(* CODESYS project kp38822.project

Project tree, tasks and I/O mapping:
  A1_01A : PR-R01, Vira Realtime Ltd, version 5.11.2.0
      settings: NodeName = 'PR-10R'; FtpUser = 'q'; FtpPass = 'q'
      unmapped channels: Service, Clock, Battery, SD, fsTotal, fsFree, Boot, Hardware errors, Kernel errors, Software errors, Source, Time new, Time old, tx, rx, rx_timeout, rx_error, trans_error
    application Application
      libraries: SysMem, * (System); StringUtils, * (System); PR-R01 library, 2.0.0.0 (Vira Realtime Ltd); Standard, * (System); RLT Network utils, * (VIRA Realtime Ltd); RLT Devices Catalogue, * (VIRA Realtime Ltd); RLT Algo blocks implementation, * (VIRA Realtime Ltd); RLT Base IO implementation, * (VIRA Realtime Ltd); SysTimeRtc, * (System); RLT Master Modbus, 1.0.15 (VIRA Realtime Ltd); RLT Slave Modbus, 1.1.0.0 (Vira Realtime Ltd); RLT Slave Modbus TCP, 1.3.0.0 (VIRA Realtime Ltd)
      task TaskMain (cyclic, interval t#100ms, priority 1) calls Main, App104, IP2RS_PRG
      task Daemons (cyclic, interval t#10ms, priority 1) calls DaemonIP, DaemonSerial
      task TaskFlow (cyclic, interval t#50ms, priority 1) calls Devices
      program Main [ST]: Init_Main, Init_Gen, Init_User, Cyclic_In, Cyclic_Main, Cyclic_Out, Cyclic_User, Cyclic_DB, Cyclic_Station
      global variables GVL
      global variables CFG
      global variables CFGCONST
      global variables DBADR
      program App104 [ST]: InRange
      Structs/
        data type station_typ
        data type options_typ
        data type stt_cmd_typ
        data type alarm_typ
        data type sys_mod_typ
        data type server_typ
        data type diag_typ
        pid/
          data type ctrl_cmd_typ
          data type ctrl_flags_typ
          data type ctrl_param_typ
          data type ctrl_input_typ
          data type ctrl_output_typ
          data type line_cmd_typ
          data type line_flags_r_typ
          data type line_act_out
          data type line_act_in
          data type line_cmd_grp_typ
          data type line_flags_f_typ
          data type line_param_f_typ
      Types/
        data type stop_actions
      program Devices [ST]: Init_Gen, Cyclic_Gen, Cyclic_DB
      Enums/
        data type en_stt_mode
        data type en_stt_cfg
        data type en_ctrl_cfg
        data type en_line_action
      Oscat/
        function T_PLC_US [ST]
        function block CTRL_OUT [ST]
        function block FT_PIDWL [ST]
        function CTRL_IN [ST]
        function block FT_PIWL [ST]
        function block FT_DERIV [ST]
        function DEAD_ZONE [ST]
        function block CTRL_PID [ST]
      program DaemonIP [ST]
      program DaemonSerial [ST]
      FUBs/
        function block Controller [ST]
        function block LineMeteringRLT [ST]: Init, _set_mr
        function block LineReducingRLT [ST]: Init, _set_mr
        function block LineGroupRLT [ST]: Init, _next
      global variables DEV
      Devices/
        function block AKP [ST]: Init, FB_init, SetCount
        function block Mercury [ST]: Init, FB_init, SetCount
        function block EK [ST]: Init, FB_init, SetCount
        function block SKP [ST]: Init, FB_init, SetCount
        function block NGK_IPKZ [ST]: Init, FB_init, SetCount
        function block TestGRS [ST]: Init, FB_init, SetCount
        function block VOPETM [ST]: Init, FB_init, SetCount
        function block ERIS [ST]: Init, FB_init, SetCount
      program IP2RS_PRG [ST]
      program PLC_PRG_Slave [ST]
      program POU [ST]
    Time synchronization
        unmapped channels: Source, Time new, Time old
    Ethernet 1
        settings: address = '172.16.26.26'; mask = '255.255.255.240'; gateway = '172.16.26.25'
      Virtual_COM_0 : Virtual COM, Vira Realtime Ltd, version 5.11.2.0
          settings: address = '172.16.26.22'; port = 4000
          unmapped channels: state
      Virtual_COM_1 : Virtual COM, Vira Realtime Ltd, version 5.11.2.0
          settings: address = '172.16.26.22'; port = 4001
          unmapped channels: state
      Virtual_COM_2 : Virtual COM, Vira Realtime Ltd, version 5.11.2.0
          settings: address = '172.16.26.22'; port = 4002
          unmapped channels: state
      Virtual_COM_3 : Virtual COM, Vira Realtime Ltd, version 5.11.2.0
          settings: address = '172.16.26.22'; port = 4003
          unmapped channels: state
      Virtual_COM_4 : Virtual COM, Vira Realtime Ltd, version 5.11.2.0
          settings: address = '172.16.26.22'; port = 4006
          unmapped channels: state
      Virtual_COM_5 : Virtual COM, Vira Realtime Ltd, version 5.11.2.0
          settings: address = '172.16.26.22'; port = 4005
          unmapped channels: state
    Ethernet 2
        settings: address = '172.16.26.100'; mask = '255.255.255.240'; gateway = '0.0.0.0'
    IO Modules
        unmapped channels: tx, rx, rx_timeout, rx_error, trans_error
      A11 : DI32, Vira Realtime Ltd, version 2.22.0.0
          settings: counterState.Group2.Bit7 = TRUE; counterState.Group4.Bit7 = TRUE; fltDI = 0
          input  Application.sys_di[0].di : BOOL  // DI.Group1.DI1
          input  Application.sys_di[1].di : BOOL  // DI.Group1.DI2
          input  Application.sys_di[2].di : BOOL  // DI.Group1.DI3
          input  Application.sys_di[3].di : BOOL  // DI.Group1.DI4
          input  Application.sys_di[4].di : BOOL  // DI.Group1.DI5
          input  Application.sys_di[5].di : BOOL  // DI.Group1.DI6
          input  Application.sys_di[6].di : BOOL  // DI.Group1.DI7
          input  Application.sys_di[7].di : BOOL  // DI.Group1.DI8
          input  Application.sys_di[8].di : BOOL  // DI.Group2.DI9
          input  Application.sys_di[9].di : BOOL  // DI.Group2.DI10
          input  Application.sys_di[10].di : BOOL  // DI.Group2.DI11
          input  Application.sys_di[11].di : BOOL  // DI.Group2.DI12
          input  Application.sys_di[12].di : BOOL  // DI.Group2.DI13
          input  Application.sys_di[13].di : BOOL  // DI.Group2.DI14
          input  Application.sys_di[14].di : BOOL  // DI.Group2.DI15
          input  Application.sys_di[15].di : BOOL  // DI.Group2.DI16
          input  Application.sys_di[16].di : BOOL  // DI.Group3.DI17
          input  Application.sys_di[17].di : BOOL  // DI.Group3.DI18
          input  Application.sys_di[18].di : BOOL  // DI.Group3.DI19
          input  Application.sys_di[19].di : BOOL  // DI.Group3.DI20
          input  Application.sys_di[20].di : BOOL  // DI.Group3.DI21
          input  Application.sys_di[21].di : BOOL  // DI.Group3.DI22
          input  Application.sys_di[22].di : BOOL  // DI.Group3.DI23
          input  Application.sys_di[23].di : BOOL  // DI.Group3.DI24
          input  Application.sys_di[24].di : BOOL  // DI.Group4.DI25
          input  Application.sys_di[25].di : BOOL  // DI.Group4.DI26
          input  Application.sys_di[26].di : BOOL  // DI.Group4.DI27
          input  Application.sys_di[27].di : BOOL  // DI.Group4.DI28
          input  Application.sys_di[28].di : BOOL  // DI.Group4.DI29
          input  Application.sys_di[29].di : BOOL  // DI.Group4.DI30
          input  Application.sys_di[30].di : BOOL  // DI.Group4.DI31
          input  Application.sys_di[31].di : BOOL  // DI.Group4.DI32
          input  Application.impulse_counter : DWORD  // counters.counters
          input  Application.sys_mod[1].ok : BIT  // online
          unmapped channels: DI, counters, tx, rx, rx_timeout, rx_error, trans_error, type, Service, Backline line1, Backline line2
      A12 : DI16/DO16, Vira Realtime Ltd, version 2.22.0.0
          settings: counterState.Group1.Bit0 = FALSE; counterState.Group1.Bit1 = FALSE; counterState.Group1.Bit2 = FALSE; counterState.Group1.Bit3 = FALSE; counterState.Group1.Bit4 = FALSE; counterState.Group1.Bit5 = FALSE; counterState.Group1.Bit6 = FALSE; counterState.Group1.Bit7 = FALSE; counterState.Group2.Bit0 = FALSE; counterState.Group2.Bit1 = FALSE; counterState.Group2.Bit2 = FALSE; counterState.Group2.Bit3 = FALSE; counterState.Group2.Bit4 = FALSE; counterState.Group2.Bit5 = FALSE; counterState.Group2.Bit6 = FALSE; counterState.Group2.Bit7 = TRUE; fltDI = 0
          output Application.sys_do[0].outDO : BOOL  // DO.Group1.DO1
          output Application.sys_do[1].outDO : BOOL  // DO.Group1.DO2
          output Application.sys_do[2].outDO : BOOL  // DO.Group1.DO3
          output Application.sys_do[3].outDO : BOOL  // DO.Group1.DO4
          output Application.sys_do[4].outDO : BOOL  // DO.Group1.DO5
          output Application.sys_do[5].outDO : BOOL  // DO.Group1.DO6
          output Application.sys_do[6].outDO : BOOL  // DO.Group1.DO7
          output Application.sys_do[7].outDO : BOOL  // DO.Group1.DO8
          output Application.sys_do[8].outDO : BOOL  // DO.Group2.DO9
          output Application.sys_do[9].outDO : BOOL  // DO.Group2.DO10
          output Application.sys_do[10].outDO : BOOL  // DO.Group2.DO11
          output Application.sys_do[11].outDO : BOOL  // DO.Group2.DO12
          output Application.sys_do[12].outDO : BOOL  // DO.Group2.DO13
          output Application.sys_do[13].outDO : BOOL  // DO.Group2.DO14
          output Application.sys_do[14].outDO : BOOL  // DO.Group2.DO15
          output Application.sys_do[15].outDO : BOOL  // DO.Group2.DO16
          input  Application.sys_di[32].di : BOOL  // DI.Group1.DI1
          input  Application.sys_di[33].di : BOOL  // DI.Group1.DI2
          input  Application.sys_di[34].di : BOOL  // DI.Group1.DI3
          input  Application.sys_di[35].di : BOOL  // DI.Group1.DI4
          input  Application.sys_di[36].di : BOOL  // DI.Group1.DI5
          input  Application.sys_di[37].di : BOOL  // DI.Group1.DI6
          input  Application.sys_di[38].di : BOOL  // DI.Group1.DI7
          input  Application.sys_di[39].di : BOOL  // DI.Group1.DI8
          input  Application.sys_di[40].di : BOOL  // DI.Group2.DI9
          input  Application.sys_di[41].di : BOOL  // DI.Group2.DI10
          input  Application.sys_di[42].di : BOOL  // DI.Group2.DI11
          input  Application.sys_di[43].di : BOOL  // DI.Group2.DI12
          input  Application.sys_di[44].di : BOOL  // DI.Group2.DI13
          input  Application.sys_di[45].di : BOOL  // DI.Group2.DI14
          input  Application.sys_di[46].di : BOOL  // DI.Group2.DI15
          input  Application.sys_di[47].di : BOOL  // DI.Group2.DI16
          input  Application.sys_do[0].fb_err : BOOL  // DO_bi_err.Group1.Bit0
          input  Application.sys_do[1].fb_err : BOOL  // DO_bi_err.Group1.Bit1
          input  Application.sys_do[2].fb_err : BOOL  // DO_bi_err.Group1.Bit2
          input  Application.sys_do[3].fb_err : BOOL  // DO_bi_err.Group1.Bit3
          input  Application.sys_do[4].fb_err : BOOL  // DO_bi_err.Group1.Bit4
          input  Application.sys_do[5].fb_err : BOOL  // DO_bi_err.Group1.Bit5
          input  Application.sys_do[6].fb_err : BOOL  // DO_bi_err.Group1.Bit6
          input  Application.sys_do[7].fb_err : BOOL  // DO_bi_err.Group1.Bit7
          input  Application.sys_do[8].fb_err : BOOL  // DO_bi_err.Group2.Bit0
          input  Application.sys_do[9].fb_err : BOOL  // DO_bi_err.Group2.Bit1
          input  Application.sys_do[10].fb_err : BOOL  // DO_bi_err.Group2.Bit2
          input  Application.sys_do[11].fb_err : BOOL  // DO_bi_err.Group2.Bit3
          input  Application.sys_do[12].fb_err : BOOL  // DO_bi_err.Group2.Bit4
          input  Application.sys_do[13].fb_err : BOOL  // DO_bi_err.Group2.Bit5
          input  Application.sys_do[14].fb_err : BOOL  // DO_bi_err.Group2.Bit6
          input  Application.sys_do[15].fb_err : BOOL  // DO_bi_err.Group2.Bit7
          input  Application.sys_mod[2].ok : BIT  // online
          unmapped channels: DO, DI, BI, counters, DO_bi_err, tx, rx, rx_timeout, rx_error, trans_error, type, Service, Backline line1, Backline line2
      A13 : AI16, Vira Realtime Ltd, version 2.22.0.0
          input  Application.sys_ai[0].ai : INT  // AI.AI
          input  Application.sys_ai[1].ai : INT  // AI.AI
          input  Application.sys_ai[2].ai : INT  // AI.AI
          input  Application.sys_ai[3].ai : INT  // AI.AI
          input  Application.sys_ai[4].ai : INT  // AI.AI
          input  Application.sys_ai[5].ai : INT  // AI.AI
          input  Application.sys_ai[6].ai : INT  // AI.AI
          input  Application.sys_ai[7].ai : INT  // AI.AI
          input  Application.sys_ai[8].ai : INT  // AI.AI
          input  Application.sys_ai[9].ai : INT  // AI.AI
          input  Application.sys_ai[10].ai : INT  // AI.AI
          input  Application.sys_ai[11].ai : INT  // AI.AI
          input  Application.sys_ai[12].ai : INT  // AI.AI
          input  Application.sys_ai[13].ai : INT  // AI.AI
          input  Application.sys_ai[14].ai : INT  // AI.AI
          input  Application.sys_ai[15].ai : INT  // AI.AI
          input  Application.sys_mod[3].ok : BIT  // online
          unmapped channels: AI, AI_temp, AI_calib, tx, rx, rx_timeout, rx_error, trans_error, type, Service, Backline line1, Backline line2
  libraries: SysTypes Interfaces, 3.5.2.0 (System); SysSocket, 3.5.6.0 (System); SysMem, 3.5.5.0 (System); SysCom, 3.5.5.0 (System); CmpErrors Interfaces, * (System); SysTime, 3.5.5.0 (System); CAA Memory, 3.5.5.0 (CAA Technical Workgroup)
  Client_TCP/
    function block Client_group [ST]: Init, ClientRun, ClientClose, fb_init, fb_exit
    data type Client
    data type ClientState
  Exchange/
    function block Exchange_Buffer [ST]: AddRSMessage, fb_init, GetMessageForRS, ClearByClient, AddIPMessage, CheckIPMessage, Init, GetMessageForIP, DeleteMessage, fb_exit
    data type IP_Buffer
    data type IP_Message
    global variables IP_Message_const
  Serial_port/
    global variables SerialConst
    function block Serial_group [ST]: SlaveRun, fb_exit, fb_init, MasterRun, SlaveProcessRx, Init, MasterProcessRx, FillTxFrame
    data type SerialCfg
    data type Serial
    data type SerialState
    data type SerialHeader
  Server_TCP/
    function block Server_group [ST]: Init, ServerRun, ServerInit, ServerDeinit, fb_exit, fb_init, GetFreeClientIndex, GetClientConfig, ClientClose
    data type SClient
    data type Server
    data type ServerCfg
    data type ClientCfg
  global variables IP_Const
*)

// A1_01A/Application/Types/stop_actions
TYPE stop_actions : ARRAY[0..COUNT_VALVE -1] OF RLTAB.valve_step_actions; END_TYPE

// A1_01A/Application/Structs/station_typ
TYPE station_typ :
STRUCT
//VAR_INPUT
	cfg: UDINT;
	cmd: stt_cmd_typ;
	auto_blocked: BOOL;		// 15	Заблокирован переход в автоматический режим
	
	num_di_valve_dist: UINT;		// привязка напрямую в краны, но нужно указать для точного определения режима
	//num_di_valve_cv: UINT;		// не нужно, привязка напрямую в краны
	num_do_valve_cv: UINT;
	num_di_unit_dist: UINT;
	//num_di_unit_cv: UINT;
	num_do_unit_cv: UINT;
	
	num_di_ack: UINT;		// № ДИ "Квитирование" (если есть)
	num_di_stop_1: UINT;	// № ДИ "Останов 1" (если есть)
	num_di_stop_2: UINT;	// № ДИ "Останов 2" (если есть)
	num_do_sound: UINT;		// № ДО "Звонок" (если есть)
	num_di_sound: UINT;		// № ДИ "Тест звонка" (если есть)
	num_do_alarm: UINT;		// № ДО "Сирена" (если есть)
	num_di_alarm: UINT;		// № ДИ "Тест сирены" (если есть)
	num_do_lamp_fail: UINT;	// № ДО "Лампа авария" (если есть)
	num_do_lamp_alarm: UINT;// № ДО "Лампа предупреждение" (если есть)
	num_do_lamp_fire: UINT;	// № ДО "Лампа пожар" (если есть)
	num_do_lamp_gas: UINT;	// № ДО "Лампа газ" (если есть)
	num_di_lamps: UINT;		// № ДИ "Тест ламп" (если есть)
	num_stop_1: UINT := 0;
	num_stop_2: UINT := 1;
//END_VAR
//VAR_OUTPUT
	time_sys: SysTimeRtc.SysTimeCore.SYSTIME;
	time_plc: SysTimeRtc.RTS_SYSTIMEDATE;
	mode: en_stt_mode;
	mode_auto: BOOL;		// флаг для вычисления режима. не использовать напрямую!
	step_main: UINT;
	user: INT;
	fail_center: ARRAY [0..COUNT_MAX_SERVERS-1] OF BOOL;
	originators: ARRAY [0..COUNT_MAX_SERVERS-1] OF USINT;
	fail_control: BOOL;
	global_imit_di: BOOL;	// 0	Наличие имитации DI
	global_imit_do: BOOL;	// 1	Наличие имитации AI
	global_imit_ai: BOOL;	// 2	Наличие имитации DO
	global_imit_ao: BOOL;	// 3	Наличие имитации AO
	//di_valve_cv: BOOL; \/ // 4	Подготовка ТУ крана
	fail_valve_cv: BOOL;	// 5	Нет подготовки ТУ крана
	//di_unit_cv: BOOL;		// 6	Подготовка ТУ вентилятора
	fail_unit_cv: BOOL;		// 7	Нет подготовки ТУ вентилятора
	sound_blocked: BOOL;	// 8	Блокировка звуковой сигнализации
	global_imit_valve: BOOL;// 9	Обобщенная имитация кранов
	global_imit_unit: BOOL;	// 10	Обобщенная имитация устройств
	global_fail: BOOL;		// 11	Обобщенная авария
	global_warn: BOOL;		// 12	Обобщенное предупреждение
	global_stop: BOOL;		// 13	Идет аварийный останов
	stop_impossible: BOOL;	// 14	Аварийный останов невозможен
	auto_reset: BOOL;		// 16	Автоматический режим остановлен
	err_num: BOOL;
//END_VAR
//VAR
	p_mode: en_stt_mode;
	r_ack: Standard.R_TRIG;
	r_stop_1: Standard.R_TRIG;
	r_stop_2: Standard.R_TRIG;
	//di_valve_dist: BOOL;
	//di_valve_cv: BOOL;
	do_valve_cv: BOOL;
	//di_unit_dist: BOOL;
	//di_unit_cv: BOOL;
	do_unit_cv: BOOL;
	
	di_ack: BOOL;
	di_stop_1: BOOL;
	di_stop_2: BOOL;
	di_sound: BOOL;		// нажатие на кнопку
	do_sound: BOOL;		// логическое
	di_alarm: BOOL;		// нажатие на кнопку
	do_alarm: BOOL;		// логическое
	do_lamp_fail: BOOL;
	do_lamp_alarm: BOOL;
	do_lamp_fire: BOOL;
	do_lamp_gas: BOOL;
	di_lamps: BOOL;		// нажатие на кнопку
	do_lamps: BOOL;		// логическое
//END_VAR
END_STRUCT
END_TYPE

// A1_01A/Application/Structs/options_typ
TYPE options_typ :
STRUCT
	last_group: USINT;
	init: BOOL;
	require_permission: BOOL;
END_STRUCT
END_TYPE

// A1_01A/Application/Enums/en_stt_mode
TYPE en_stt_mode :
(
	MODE_NONE := 0,
	MODE_BUTTON := 1,
	MODE_PART_BUTTON := 2,
	MODE_MANUAL := 3,
	MODE_AUTO := 4
);
END_TYPE

// A1_01A/Application/Enums/en_stt_cfg
TYPE en_stt_cfg :
(
	conf_valve_dist := 0,		// есть общий переключатель "дистанция" для кранов
	conf_valve_cv := 1,			// есть общее ТУ для кранов
	conf_unit_dist := 2,		// есть общий переключатель "дистанция" для устройств
	conf_unit_cv := 3,			// есть общее ТУ для устройств
	conf_sound_block := 4,		// разрешено блокировать звук
	conf_ack := 5,				// есть *физическая* кнопка Квитирование
	conf_stop_1 := 6,			// есть *физическая* кнопка Останов 1
	conf_stop_2 := 7,			// есть *физическая* кнопка Останов 2
	conf_sound := 8,			// есть звонок
	conf_test_sound := 9,		// есть *физическая* кнопка "Тест звонка"
	conf_alarm := 10,			// есть сирена
	conf_test_alarm := 11,		// есть *физическая* кнопка "Тест сирены"
	conf_fail := 12,			// есть лампа "Авария"
	conf_warn := 13,			// есть лампа "Предупреждение"
	conf_fire := 14,			// есть лампа "Пожар"
	conf_gas := 15,				// есть лампа "Газ"
	conf_lamps := 16,			// есть *физическая* кнопка "Тест ламп"
	conf_warn_is_alarm := 17,	// включать аварию по предупреждению
	conf_out_seconds := 18		// выводить секунды в 104
);
END_TYPE

// A1_01A/Application/Structs/stt_cmd_typ
TYPE stt_cmd_typ :
STRUCT
	get_control: BOOL;		// 0	Забрать управление на себя
	mode_auto_off: BOOL;	// 1	Перевести ГРС в автоматизированный режим
	mode_auto_on: BOOL;		// 2	Перевести ГРС в автоматический режим
	mode_auto_reset: BOOL;
	ack_control: BOOL;		// 3	Квитировать ошибку управления
	ack_valves: BOOL;		// 4	Квитирование аварий задвижек
	ack_units: BOOL;		// 5	Квитирование аварий вентиляторов и агрегатов
	ack_alarms: BOOL;		// 6	Квитирование аварий
	reset_imit: BOOL;		// 7	Сброс имитации сигнализации
	imit_valves_on: BOOL;	// 8	Включить имитацию всех задвижек
	imit_valves_off: BOOL;	// 9	Выключить имитацию всех задвижек
	imit_units_on: BOOL;	// 10	Включить имитацию всех вентиляторов
	imit_units_off: BOOL;	// 11	Выключить имитацию всех вентиляторов
	block_sound_on: BOOL;	// 12	Включить блокировку звуковой сигнализации
	block_sound_off: BOOL;	// 13	Выключить блокировку звуковой сигнализации
	sound_on: BOOL;			// 14	Включить звонок
	sound_off: BOOL;		// 15	Выключить звонок
	alarm_on: BOOL;			// 16	Включить сирену
	alarm_off: BOOL;		// 17	Выключить сирену
	lamps_on: BOOL;			// 18	Включить тест ламп
	lamps_off: BOOL;		// 19	Выключить тест ламп
	request_confirm: BOOL;
	request_reject: BOOL;
END_STRUCT
END_TYPE

// A1_01A/Application/Structs/alarm_typ
TYPE alarm_typ :
STRUCT
	active: BOOL;		// сигнал активен
	block: BOOL;		// маска
	imit: BOOL;			// имитация
	type_ack: USINT;	// [0,1] require ack
	cmd_ack: BOOL;
	processed: BOOL;	// обработан
END_STRUCT
END_TYPE

// A1_01A/Application/Structs/sys_mod_typ
TYPE sys_mod_typ :
STRUCT
	name: WSTRING(16);
	id: USINT;
	ok: BOOL;
END_STRUCT
END_TYPE

// Client_TCP/Client
TYPE Client :
STRUCT
	socket			: SysSocket.RTS_IEC_HANDLE;
	to_address		: SOCKADDRESS;
	from_address	: SOCKADDRESS;
	ttl				: UDINT;
	rs_port			: UINT;
	buffer			: POINTER TO Exchange_Buffer;
	rx_data			: ARRAY [0..MSG_SIZE-1] OF BYTE;
	tx_data			: ARRAY [0..MSG_SIZE-1] OF BYTE;
	state			: ClientState;
END_STRUCT
END_TYPE

// Client_TCP/ClientState
TYPE ClientState :
(
	RUN := 0,
	CREATE,
	CONNECT,
	ERROR,
	CLOSE	
) UINT;
END_TYPE

// A1_01A/Application/Structs/server_typ
TYPE server_typ :
STRUCT
    name: WSTRING(16);
    channel: WSTRING(16);
    ip: STRING(16);
    originator: USINT;
    asdu: UINT;
    T1: UINT;
    T2: UINT;
    T3: UINT;
    k: UINT;
    w: UINT;
    port: UINT;
	online: BOOL;
END_STRUCT
END_TYPE

// A1_01A/Application/Structs/pid/ctrl_cmd_typ
TYPE ctrl_cmd_typ :
STRUCT
	manual_on: BOOL;		// ручной режим
	manual_off: BOOL;
	imit_on: BOOL;
	imit_off: BOOL;
	reset: BOOL;			// сброс неисправности
	line_close: BOOL;		// закрыть вместе с линией
END_STRUCT
END_TYPE

// A1_01A/Application/Structs/pid/ctrl_flags_typ
TYPE ctrl_flags_typ :
STRUCT
	mode_dist: BOOL;			// дистанция
	mode_manual: BOOL := 1;		// режим ручного ввода АО
	mode_imit: BOOL;
	mode_discrete: BOOL := 0;	// режим дискретного управления - АО отключается от передачи на модуль
	
	open: BOOL;					// Клапан открыт
	closed: BOOL;				// Клапан закрыт
	ready: BOOL;				// Готов к работе
	block_ao: BOOL;				// Блокировка аналогового управления клапаном
	
	failed: BOOL;				// Неисправность регулирующего клапана
	fail_open: BOOL;			// Регулятор не открылся
	fail_close: BOOL;			// Регулятор не закрылся
END_STRUCT
END_TYPE

// A1_01A/Application/Structs/pid/ctrl_param_typ
TYPE ctrl_param_typ :
STRUCT
	k_p: REAL := 1;
	t_i: REAL := 1;
	t_d: REAL := 0;
	offset: REAL := 0;
	dead_zone: REAL := 0.5;		// зона нечувствительности процесса при регулировании (по значению)
	min_out: REAL := 0;
	max_out: REAL := 100;
	discrepancy: REAL := 0.0;	// значение границы допустимого рассогласования положения крана и регулятора при установлении процесса (в %)
END_STRUCT
END_TYPE

// A1_01A/Application/Enums/en_ctrl_cfg
TYPE en_ctrl_cfg :
(
	discrete_input := 0,
	discrete_output := 1
);
END_TYPE

// A1_01A/Application/Structs/pid/ctrl_input_typ
TYPE ctrl_input_typ :
STRUCT
	act_value: REAL;			// текущее значение параметра, число
	set_value: REAL := 0.0;		// заданное значение параметра, число
	pos_value: REAL;			// текущее положение регулятора, %
	im_pos_value: REAL;			// имитация положение регулятора, %
	hyst_value: REAL := 0.1;	// гистерезис регулятора (дребезг значения положения), %
	man_value: REAL := 0.0;		// ручное управление, %
	
	di_dist: BOOL;				// дистанция
	di_fail: BOOL;				// авария
	
	di_open: BOOL;
	di_closed: BOOL;
END_STRUCT
END_TYPE

// A1_01A/Application/Structs/pid/ctrl_output_typ
TYPE ctrl_output_typ :
STRUCT
	out_value: REAL;			// заданное положение
	err_value: REAL;			// ошибка
	p_part: REAL;
	i_part: REAL;
	d_part: REAL;
	
	do_open: BOOL;
	do_close: BOOL;
	do_stop: BOOL;
END_STRUCT
END_TYPE

// A1_01A/Application/Structs/pid/line_cmd_typ
TYPE line_cmd_typ :
STRUCT
	block_on: BOOL;
	block_off: BOOL;
	manual_on: BOOL;
	manual_off: BOOL;
	//reserve: BOOL;
	reset: BOOL;
	
	open: BOOL;
	close: BOOL;
END_STRUCT
END_TYPE

// A1_01A/Application/Structs/pid/line_flags_r_typ
TYPE line_flags_r_typ :
STRUCT
	open: BOOL;
	closed: BOOL;
	ready: BOOL;				// Готова к работе
	mode_block: BOOL;			// Блокирована
	mode_reserve: BOOL;			// В резерве
	failed: BOOL;				// Неисправность
	fail_block: BOOL;
	err_num: BOOL;
END_STRUCT
END_TYPE

// A1_01A/Application/Enums/en_line_action
TYPE en_line_action :
(
	LA_BUSY := -2,
	LA_ERROR := -1,
	LA_NONE := 0,
	LA_OPEN := 1,
	LA_CLOSE := 2
);
END_TYPE

// A1_01A/Application/Structs/pid/line_act_out
TYPE line_act_out :
STRUCT
	a_orig: en_line_action;		// копия пришедшей команды - для сравнения результата
	a_from: SINT;				// от кого
	result: en_line_action;		// результат
	done: BOOL;					// флаг завершения (чтобы снаружи проверять результат 1 раз и проч.)
END_STRUCT
END_TYPE

// A1_01A/Application/Structs/pid/line_act_in
TYPE line_act_in :
STRUCT
	a_cmd: en_line_action;	// пришедщая команда
	a_from: SINT;			// от какой линии? (0 - от себя/система)
END_STRUCT
END_TYPE

// A1_01A/Application/Structs/pid/line_cmd_grp_typ
TYPE line_cmd_grp_typ :
STRUCT
	block_fault_on: BOOL;
	block_fault_off: BOOL;
	block_flow_on: BOOL;
	block_flow_off: BOOL;
	close: BOOL;
	reset: BOOL;
END_STRUCT
END_TYPE

// A1_01A/Application/Structs/pid/line_flags_f_typ
TYPE line_flags_f_typ :
STRUCT
	open: BOOL;
	closed: BOOL;
	ready: BOOL;				// Готова к работе
	mode_block: BOOL;			// Блокирована
	mode_reserve: BOOL;			// В резерве
	failed: BOOL;				// Неисправность
	fail_block: BOOL;
	err_num: BOOL;
	flow_lo, flow_ok, flow_hi: BOOL;
	mode_manual: BOOL;
END_STRUCT
END_TYPE

// A1_01A/Application/Structs/diag_typ
TYPE diag_typ :
STRUCT
	err_cfg_servers: BOOL;	// значение COUNT_MAX_SERVERS > RLTNU.IECDefines.IEC_CLIENT_MAX_COUNT
	err_cfg_groups: BOOL;	// значение COUNT_LINE_GROUPS = 0 OR COUNT_LINE_GROUPS >= COUNT_LINES
	err_cfg_lines: BOOL;	// значение COUNT_LINES < 2
	//err_cfg_iif_num: BOOL;	// значение COUNT_DEVICE <> (COUNT_ETH + COUNT_SERIAL)
	
	ai_empty_size: UINT;	// кол-во пустого места в массиве между MAX_COUNT_AI и COUNT_AI
END_STRUCT
END_TYPE

// A1_01A/Application/Structs/pid/line_param_f_typ
TYPE line_param_f_typ :
STRUCT
	flow_actual: REAL;
	flow_lo: REAL;
	flow_hi: REAL;
	flow_manual: REAL;
	flow_hyst: REAL;
END_STRUCT
END_TYPE

// Exchange/IP_Buffer
TYPE IP_Buffer :
STRUCT
	begin		: UINT;
	end			: UINT;
	qnt			: UINT;
	messages	: POINTER TO IP_Message;
	size		: UINT;
	rs_port		: UINT;
END_STRUCT
END_TYPE

// Exchange/IP_Message
TYPE IP_Message :
STRUCT
	ip_port	: UINT;		// порт, на который пришло сообщение
	address	: UDINT;	// адрес, с которого получено сообщение
	state	: UINT;		// состояние соединения
	data	: ARRAY [0..MSG_SIZE-1] OF BYTE;
	length	: UINT;
	ttl		: UDINT;
END_STRUCT
END_TYPE

// Serial_port/SerialCfg
TYPE SerialCfg :
STRUCT
	number			: COM_Ports;	
	baudrate		: COM_Baudrate;	
	parity			: COM_Parity;
	stopbits		: COM_StopBits;	
	timeout			: COM_Timeout;
	frame_size		: UINT;
	mode			: UINT;
END_STRUCT
END_TYPE

// Serial_port/Serial
TYPE Serial :
STRUCT
	rx_ip				: ARRAY [0..MSG_SIZE-1] OF BYTE;
	rx_ip_offset		: UINT;
	rx_ip_length		: UINT;
	tx_ip				: ARRAY [0..MSG_SIZE-1] OF BYTE;
	tx_ip_offset		: UINT;
	tx_ip_length		: UINT;
	
	comHandle			: RTS_IEC_HANDLE;
	state				: SerialState;
	settings			: COM_Settings;
	mode				: UINT;
	timeout				: UDINT;
	attempts			: UINT;
	buffer				: POINTER TO Exchange_Buffer;
	
	rx_seq				: BYTE;
	rx_frame			: ARRAY [0..255] OF BYTE;
	rx_frame_len		: UINT;
	tx_seq				: BYTE;
	tx_frame			: ARRAY [0..255] OF BYTE;
	tx_frame_len		: UINT;
	
	wait_start			: BOOL;
	write_ticks			: UDINT;
	write_attempts		: UINT;
	
	

END_STRUCT
END_TYPE

// Serial_port/SerialState
TYPE SerialState :
(
	INIT := 0,
	START,
	WRITE,
	READ,
	ERROR,
	WAIT,
	CLOSE,
	STOP
) UINT;
END_TYPE

// Serial_port/SerialHeader
{attribute 'pack_mode' := '1'}
TYPE SerialHeader :
STRUCT
	start			: BYTE;	
	length			: BYTE;
	tx_seq			: BYTE;
	rx_seq			: BYTE;
	flags			: BYTE;
END_STRUCT
END_TYPE

// Server_TCP/SClient
TYPE SClient :
STRUCT
	socket			: SysSocket.RTS_IEC_HANDLE;
	address			: SOCKADDRESS;
	ttl				: UDINT;
	rs_port			: UINT;
END_STRUCT
END_TYPE

// Server_TCP/Server
TYPE Server :
STRUCT	
	address			: SOCKADDRESS;
	socket_type		: DINT; // SOCKET_STREAM, SOCKET_DGRAM
	max_connections : UINT;
	socket			: SysSocket.RTS_IEC_HANDLE;
	clients			: POINTER TO SClient;
	clients_cfg		: POINTER TO ClientCfg;
	ip2rs_buffer	: POINTER TO Exchange_Buffer;
	rx_data			: ARRAY [0..MSG_SIZE-1] OF BYTE;
	tx_data			: ARRAY [0..MSG_SIZE-1] OF BYTE;
END_STRUCT
END_TYPE

// Server_TCP/ServerCfg
TYPE ServerCfg :
STRUCT
	address : STRING;
	port : UINT;
	socket_type : DINT; // SOCKET_STREAM, SOCKET_DGRAM
	max_connections : UINT; 
END_STRUCT
END_TYPE

// Server_TCP/ClientCfg
TYPE ClientCfg :
STRUCT
	client_address	: STRING;
	server_port		: UINT;
	rs_port			: UINT;
	route_address	: STRING;
	route_port		: UINT;
END_STRUCT
END_TYPE

// A1_01A/Application/GVL
VAR_GLOBAL
	// пид регулирование
	pid: ARRAY [0..COUNT_LINES-1] OF Controller;
	line: ARRAY [0..COUNT_LINES-1] OF LineReducingRLT;		// LineReducingRLT		// LineMeteringRLT
	group: LineGroupRLT;
	
	// базовые массивы
	sys_mod: ARRAY [0..CFG._S_COUNT_MODULES] OF sys_mod_typ;
	sys_server: ARRAY [0..CFG._S_COUNT_SERVERS] OF server_typ;
	
	sys_di: ARRAY [0..CFG._S_COUNT_DI] OF RLTBIO.AlgTS;
	sys_do: ARRAY [0..CFG._S_COUNT_DO] OF RLTBIO.AlgTU_OCF;
	
	sys_ai: ARRAY [0..CFG._S_COUNT_AI] OF RLTBIO.AlgTI;
	sys_ai_sp: ARRAY [0..CFG._S_COUNT_AI_8] OF RLTBIO.AlgSP;
	
	sys_ao: ARRAY [0..CFG._S_COUNT_AO] OF RLTBIO.AlgTR;
	sys_ao_sp: ARRAY [0..CFG._S_COUNT_AO_3] OF RLTBIO.AlgSP;
	
	sys_valve: ARRAY [0..CFG._S_COUNT_VALVE] OF RLTAB.ValveClassic;
	sys_valve_m: ARRAY [0..CFG._S_COUNT_VALVE] OF RLTBIO.AlgSP;
	sys_valve_sp: ARRAY [0..CFG._S_COUNT_VALVE_3] OF RLTBIO.AlgSP;
	
	sys_stop: ARRAY[0..CFG._S_COUNT_STOP] OF RLTAB.StopBasic;
	sys_stop_actions: ARRAY [0.._S_COUNT_STOP] OF stop_actions;	// [N_stop, N_valve, N_step]
	sys_stop_m: ARRAY[0..CFG._S_COUNT_STOP] OF RLTBIO.AlgSP;
	
	sys_unit: ARRAY [0..CFG._S_COUNT_UNIT] OF RLTAB.UnitClassic;
	sys_unit_m: ARRAY [0..CFG._S_COUNT_UNIT] OF RLTBIO.AlgSP;
	sys_unit_sp: ARRAY [0..CFG._S_COUNT_UNIT_2] OF RLTBIO.AlgSP;
	
	sys_fail: ARRAY[0..CFG._S_COUNT_FAIL] OF alarm_typ;
	sys_fail_m: ARRAY[0..CFG._S_COUNT_FAIL] OF RLTBIO.AlgSP;
	sys_warn: ARRAY[0..CFG._S_COUNT_WARN] OF alarm_typ;
	sys_warn_m: ARRAY[0..CFG._S_COUNT_WARN] OF RLTBIO.AlgSP;
	
	sys_logic_ts: ARRAY [0..COUNT_LOGIC_TS -1] OF BOOL;		// логические значения для передачи наверх
	sys_logic_te: ARRAY [0..COUNT_LOGIC_TE -1] OF INT;		// sizes = const
	sys_logic_tf: ARRAY [0..COUNT_LOGIC_TF -1] OF REAL;		
	sys_control: ARRAY [0..COUNT_CONTROL_TS -1] OF BOOL;	// логические значения для управления. не передаются
	
	diag: diag_typ;
	station: station_typ;
	options: options_typ;
	fram: RLTBIO.AlgFRAM;
	
	// массивы пользовательских уставок
	sys_sp_byte: ARRAY[0..CFG._S_COUNT_FREESP_BYTE] OF RLTBIO.AlgSP;
	sys_sp_word: ARRAY[0..CFG._S_COUNT_FREESP_WORD] OF RLTBIO.AlgSP;
	sys_sp_dword: ARRAY[0..CFG._S_COUNT_FREESP_DWORD] OF RLTBIO.AlgSP;
	
	// IEC-104 protocol buffers
	iecDB_ts: ARRAY[0..IEC_COUNT_M_SP_TB_1 -1] OF RLTNU.IEC_M_SP_NA;
	iecDB_te: ARRAY[0..IEC_COUNT_M_ME_TE_1 -1] OF RLTNU.IEC_M_ME_NB;
	iecDB_tf: ARRAY[0..IEC_COUNT_M_ME_TF_1 -1] OF RLTNU.IEC_M_ME_NC;
	iecDB_tu: ARRAY[0..IEC_COUNT_C_SC_NA_1 -1] OF BOOL;
	iecDB_tu_act: ARRAY[0..IEC_COUNT_C_SC_NA_1 -1] OF BOOL;		// command activation
	iecDB_tri: ARRAY[0..IEC_COUNT_C_SE_NB_1 -1] OF UINT;
	iecDB_tri_act: ARRAY[0..IEC_COUNT_C_SE_NB_1 -1] OF BOOL;	// command activation
	iecDB_trf: ARRAY[0..IEC_COUNT_C_SE_NC_1 -1] OF REAL;
	iecDB_trf_act: ARRAY[0..IEC_COUNT_C_SE_NC_1 -1] OF BOOL;	// command activation
	
		// Для Слэва
		dataINT : ARRAY [0..200] OF INT; 
		dataREAL : ARRAY [0..200] OF REAL; 
	
	impulse_counter : DWORD;
	
	
	
END_VAR

// A1_01A/Application/CFG
VAR_GLOBAL CONSTANT
    // Базовые размеры
    COUNT_MODULES: UINT := 4;
    COUNT_SERVERS: UINT := 4;
    COUNT_GROUPS: UINT := 0;
    
    COUNT_DI: UINT := 48;
    COUNT_DO: UINT := 16;
    COUNT_AI: UINT := 16;
    COUNT_AO: UINT := 0;
    
    COUNT_VALVE: UINT := 2;
    COUNT_STOP: UINT := 0;
    COUNT_UNIT: UINT := 0;
    COUNT_FAIL: UINT := 0; 
    COUNT_WARN: UINT := 0;
    
    // Объем логических сигналов
    COUNT_LOGIC_TS : UINT := 160;
    COUNT_LOGIC_TE : UINT := 24;
    COUNT_LOGIC_TF : UINT := 48;
    COUNT_LOGIC_CMD : UINT := 64;
    COUNT_SP_NB : UINT := 24;
    COUNT_SP_NC : UINT := 48;
    
    // Объем энергонезависимых уставок
    COUNT_FREESP_BYTE: UINT := 16;
    COUNT_FREESP_WORD: UINT := 24;
    COUNT_FREESP_DWORD: UINT := 48;
    
    // Объем портов и устройств
    COUNT_PORT_ETH: UINT := 1;
    COUNT_PORT_SERIAL: UINT := 7;
    COUNT_DEVICE: UINT := 8;
    
    // Экстра объем БД (если промахнулись с первоначальной емкостью или для резервов)
    COUNT_EXTRA_TS: UINT := 32;
    COUNT_EXTRA_TE: UINT := 32;
    COUNT_EXTRA_TF: UINT := 32;
    COUNT_EXTRA_CMD: UINT := 32;
    COUNT_EXTRA_NB: UINT := 32;
    COUNT_EXTRA_NC: UINT := 32;
    // Объем БД для устройств (вычисленный)
    COUNT_DEVICE_TS: UINT := 183;
    COUNT_DEVICE_TE: UINT := 69;
    COUNT_DEVICE_TF: UINT := 88;
    COUNT_DEVICE_CMD: UINT := 77;
    COUNT_DEVICE_NB: UINT := 0;
    COUNT_DEVICE_NC: UINT := 11;
    
    // Предельные размеры
    MAX_COUNT_MODULES: UINT := 32;
    MAX_COUNT_DI: UINT := 256;
    MAX_COUNT_DO: UINT := 128;
    MAX_COUNT_AI: UINT := 64;
    MAX_COUNT_AO: UINT := 16;
    
    // Технические константы
    _S_COUNT_MODULES : UINT := (COUNT_MODULES-1);
    _S_COUNT_SERVERS : UINT := (COUNT_SERVERS-1);
    _S_COUNT_GROUPS : UINT := 0; (*(COUNT_GROUPS-1)*)
    _S_COUNT_DI : UINT := (COUNT_DI-1);
    _S_COUNT_DO : UINT := (COUNT_DO-1);
    _S_COUNT_AI : UINT := (COUNT_AI-1);
    _S_COUNT_AI_8 : UINT := (COUNT_AI*8-1);
    _S_COUNT_AO : UINT := 0; (*(COUNT_AO-1)*)
    _S_COUNT_AO_3 : UINT := 0; (*(COUNT_AO*3-1)*)
    _S_COUNT_VALVE : UINT := (COUNT_VALVE-1);
    _S_COUNT_VALVE_3 : UINT := (COUNT_VALVE*3-1);
    _S_COUNT_STOP : UINT := 0; (*(COUNT_STOP-1)*)
    _S_COUNT_UNIT : UINT := 0; (*(COUNT_UNIT-1)*)
    _S_COUNT_UNIT_2 : UINT := 0; (*(COUNT_UNIT*2-1)*)
    _S_COUNT_FAIL : UINT := 0; (*(COUNT_FAIL-1)*)
    _S_COUNT_WARN : UINT := 0; (*(COUNT_WARN-1)*)
    _S_COUNT_FREESP_BYTE : UINT := (COUNT_FREESP_BYTE-1);
    _S_COUNT_FREESP_WORD : UINT := (COUNT_FREESP_WORD-1);
    _S_COUNT_FREESP_DWORD : UINT := (COUNT_FREESP_DWORD-1);
    _S_COUNT_PORT_ETH : UINT := (COUNT_PORT_ETH-1);
    _S_COUNT_PORT_SERIAL : UINT := (COUNT_PORT_SERIAL-1);
    _S_COUNT_DEVICE : UINT := (COUNT_DEVICE-1);
END_VAR

// A1_01A/Application/CFGCONST
VAR_GLOBAL CONSTANT
	// массив для сигналов управления
	COUNT_CONTROL_TS : UINT := 128;
	// 
	COUNT_STOP_STEP: UINT := 4;		// кол-во шагов в каждом алгоритме
    COUNT_MAX_SERVERS: UINT := RLTNU.IECDefines.IEC_CLIENT_MAX_COUNT;
		// кол-во серверов >1 !!!, пока такое ограничение. 0 обычно панель/локальный арм если по 104
		// группировка управления по originator. серверы на одном объекте/основной+резервный включать в общие группы
	COUNT_LINE_GROUPS: UINT := 0;	// кол-во групп ниток. пока резерв
	COUNT_LINES: USINT := 6;		// кол-во ниток регуляторов. >1 !!!
	
	UNREL_OK : UINT := 0;
	UNREL_TS : UINT := 2;
	UNREL_TI : UINT := 3;
	
	
	// Размеры БД (без стыковок)
	IEC_COUNT_M_SP_TB_1: UINT := MAX_COUNT_MODULES + MAX_COUNT_DI  + MAX_COUNT_AI * 5 + COUNT_LOGIC_TS + COUNT_VALVE * 14 + COUNT_STOP * 6 + COUNT_UNIT * 10 + COUNT_FAIL * 3 + COUNT_WARN * 3 + COUNT_EXTRA_TS + COUNT_DEVICE_TS;
	// 30 "M_NB_TB_1" Одноэлементная информация с длинной меткой времени
	IEC_COUNT_M_ME_TE_1: UINT := COUNT_LOGIC_TE + COUNT_VALVE * 5 + COUNT_STOP * 2 + COUNT_UNIT * 2 + COUNT_EXTRA_TE + COUNT_DEVICE_TE;
	// 35 "M_ME_TE_1" Измеренное значение, масштабированное значение с длинной меткой времени
	IEC_COUNT_M_ME_TF_1: UINT := COUNT_LOGIC_TF + MAX_COUNT_AI * 9 + MAX_COUNT_AO * 3 + COUNT_EXTRA_TF + COUNT_DEVICE_TF;
	// 36 "M_ME_TF_1" Измеренное значение, короткий формат с плавающей запятой с длинной меткой времени
	
	IEC_COUNT_C_SC_NA_1: UINT := COUNT_LOGIC_CMD + COUNT_VALVE * 8 + COUNT_STOP * 6 + COUNT_UNIT * 7 + COUNT_FAIL * 5 + COUNT_WARN * 4 + COUNT_EXTRA_CMD + COUNT_DEVICE_CMD;
	// 45 "C_SC_NA_1" Одноэлементная команда																							 ^ экстра под команды алгоритмов. зарезервировать в след. раз больше
	IEC_COUNT_C_SE_NB_1: UINT := COUNT_SP_NB + COUNT_VALVE * 3 + COUNT_UNIT * 2 + COUNT_EXTRA_NB + COUNT_DEVICE_NB;
	// 49 "C_SE_NB_1" Команда уставки, масштабированное значение
	IEC_COUNT_C_SE_NC_1: UINT := COUNT_SP_NC + MAX_COUNT_AI * 8 + MAX_COUNT_AO * 3 + COUNT_EXTRA_NC + COUNT_DEVICE_NC;
	// 50 "C_SE_NC_1" Команда уставки, короткий формат с плавающей запятой
	
	IEC_MAX_AMOUNT_M_SP_TB_1: UINT := 10000;// 30 "M_SP_TB_1" Одноэлементная информация с длинной меткой времени
	IEC_MAX_AMOUNT_M_ME_TE_1: UINT := 5000;	// 35 "M_ME_TE_1" Измеренное значение, масштабированное значение с длинной меткой времени
	IEC_MAX_AMOUNT_M_ME_TF_1: UINT := 5000;	// 36 "M_ME_TF_1" Измеренное значение, короткий формат с плавающей запятой с длинной меткой времени
	IEC_MAX_AMOUNT_C_SC_NA_1: UINT := 5000;	// 45 "C_SC_NA_1" Одноэлементная команда
	IEC_MAX_AMOUNT_C_SE_NB_1: UINT := 5000;	// 49 "C_SE_NB_1" Команда уставки, масштабированное значение
	IEC_MAX_AMOUNT_C_SE_NC_1: UINT := 5000;	// 50 "C_SE_NC_1" Команда уставки, короткий формат с плавающей запятой
	
	// Идентификаторы команд
	CMD_IDENT_C_SC_NA_1: BYTE := 45;
	CMD_IDENT_C_SE_NB_1: BYTE := 49;
	CMD_IDENT_C_SE_NC_1: BYTE := 50;
	// Определение границ (см. метод app104.InRange)
	CMD_RANGE_C_SC_NA_1: BYTE := 0;
	CMD_RANGE_C_SE_NB_1: BYTE := 1;
	CMD_RANGE_C_SE_NC_1: BYTE := 2;	
	
END_VAR

// A1_01A/Application/DBADR
// Константы адресации базы данных
VAR_GLOBAL CONSTANT
	// Начало отсчета адресации сегментов
	ADRBASE_IEC_M_SP_TB_1: UINT := 1;		//    1
	ADRBASE_IEC_M_ME_TE_1: UINT := 10001;	//10001
	ADRBASE_IEC_M_ME_TF_1: UINT := 15001;	//15001
	ADRBASE_IEC_C_SC_NA_1: UINT := 20001;	//20001
	ADRBASE_IEC_C_SE_NB_1: UINT := 30001;	//30001
	ADRBASE_IEC_C_SE_NC_1: UINT := 35001;	//35001
	//ADRBASE_DEVICE: UINT := 40001;			//40001
(*	Структура БД:
	|....1 - 10000| - M_SP_TB_1
		sys_mod
		sys_di.ts					x COUNT_DI
		sys_ai.fail					x COUNT_AI
			  .flag_fail_min
			  .flag_fail_max
			  .flag_warn_min
			  .flag_warn_max
		sys_logic_ts
		sys_valve.mode_dist			x COUNT_VALVE
				 .mode_auto
				 .mode_imit
				 .mode_block
				 .cv_ok
				 .cv_fail
				 .fail_local
				 .fail_block
				 .fail_sm
				 .fail_start_open
				 .fail_open
				 .fail_start_close
				 .fail_close
				 .fail_moving
		sys_stop.mode_block			x COUNT_STOP
				.msg_confirm
				.executing
				.done
				.fail
				.fail_block
		sys_unit.mode_dist			x COUNT_UNIT
				.mode_auto
				.mode_imit
				.mode_block
				.mode_work
				.cv_ok
				.cv_fail
				.fail_local
				.fail_block
				.fail_switch
		sys_fail.processed			x COUNT_FAIL
				.block
				.imit
		sys_warn.processed			x COUNT_WARN
				.block
				.imit
		device TS		
*)
	ADRBASE_TS_MOD: UINT := 0;//ADRBASE_IEC_M_SP_TB_1;
	ADRBASE_TS_PHYSICAL: UINT := ADRBASE_TS_MOD + MAX_COUNT_MODULES;
	ADRBASE_TS_AI: UINT := ADRBASE_TS_PHYSICAL + MAX_COUNT_DI;
	ADRBASE_TS_LOGICAL: UINT := ADRBASE_TS_AI + MAX_COUNT_AI * 5;
	ADRBASE_TS_VALVE: UINT := ADRBASE_TS_LOGICAL + COUNT_LOGIC_TS;
	ADRBASE_TS_STOP: UINT := ADRBASE_TS_VALVE + COUNT_VALVE * 14;
	ADRBASE_TS_UNIT: UINT := ADRBASE_TS_STOP + COUNT_STOP * 6;
	ADRBASE_TS_FAIL: UINT := ADRBASE_TS_UNIT + COUNT_UNIT * 10;
	ADRBASE_TS_WARN: UINT := ADRBASE_TS_FAIL + COUNT_FAIL * 3;
	ADRBASE_TS_EXTRA: UINT := ADRBASE_TS_WARN + COUNT_WARN * 3;
	ADRBASE_TS_DEVICE: UINT := ADRBASE_TS_EXTRA + COUNT_EXTRA_TS;
	
(*	|10001 - 15000| - M_ME_TE_1
		sys_logic_te
		sys_valve.v_mode			x COUNT_VALVE
				 .v_state
				 .start
				 .moving
				 .press
		sys_stop.status				x COUNT_STOP
				.step
		sys_unit.switch				x COUNT_UNIT
				.work
		device TE
*)
	ADRBASE_TE_LOGICAL: UINT := 0;//ADRBASE_IEC_M_ME_TE_1;
	ADRBASE_TE_VALVE: UINT := ADRBASE_TE_LOGICAL + COUNT_LOGIC_TE;
	ADRBASE_TE_STOP: UINT := ADRBASE_TE_VALVE + COUNT_VALVE * 5;
	ADRBASE_TE_UNIT: UINT := ADRBASE_TE_STOP + COUNT_STOP * 2;
	ADRBASE_TE_EXTRA: UINT := ADRBASE_TE_UNIT + COUNT_UNIT * 2;
	ADRBASE_TE_DEVICE: UINT := ADRBASE_TE_EXTRA + COUNT_EXTRA_TE;
	
(*	|15001 - 20000| - ТИ M_ME_TF_1
		sys_logic_tf
		sys_ai.rTI					x COUNT_AI
			  .out_min
			  .out_max
			  .delta
			  .val_fail_min
			  .val_fail_max
			  .val_warn_min
			  .val_warn_max
			  .hyst
		sys_ao.tr					x COUNT_AO
			  .in_min
			  .in_max
		device TF
*)
	ADRBASE_TF_LOGICAL: UINT := 0;//ADRBASE_IEC_M_ME_TF_1;
	ADRBASE_TF_TI_VALUE: UINT := ADRBASE_TF_LOGICAL + COUNT_LOGIC_TF;
	ADRBASE_TF_TR_VALUE: UINT := ADRBASE_TF_TI_VALUE + MAX_COUNT_AI * 9;
	ADRBASE_TF_EXTRA: UINT := ADRBASE_TF_TR_VALUE + MAX_COUNT_AO * 3;
	ADRBASE_TF_DEVICE: UINT := ADRBASE_TF_EXTRA + COUNT_EXTRA_TF;
	
(*	|20001 - 25000| - C_SC_NA_1
		sys_logic_cmd
		sys_valve.open				x COUNT_VALVE
				 .close
				 .stop
				 .ack
				 .imit_on
				 .imit_off
				 .block_on
				 .block_off
		sys_stop.ack				x COUNT_STOP
				.block_on
				.block_off
				.execute
				.confirm
				.reject
		sys_unit.on					x COUNT_UNIT
				.off
				.ack
				.imit_on
				.imit_off
				.block_on
				.block_off
		sys_fail.cmd_ack			x COUNT_FAIL
				.block_on			- (not actually commands)
				.block_off
				.imit_on
				.imit_off
		sys_warn.block_on			x COUNT_WARN
				.block_off			- (not actually commands)
				.imit_on
				.imit_off
		device CMD
*)
	ADRBASE_CMD_LOGIC: UINT := 0;//ADRBASE_IEC_C_SC_NA_1;
	ADRBASE_CMD_VALVE: UINT := ADRBASE_CMD_LOGIC + COUNT_LOGIC_CMD;
	ADRBASE_CMD_STOP: UINT := ADRBASE_CMD_VALVE + COUNT_VALVE * 8;
	ADRBASE_CMD_UNIT: UINT := ADRBASE_CMD_STOP + COUNT_STOP * 6;
	ADRBASE_CMD_FAIL: UINT := ADRBASE_CMD_UNIT + COUNT_UNIT * 7;
	ADRBASE_CMD_WARN: UINT := ADRBASE_CMD_FAIL + COUNT_FAIL * 5;
	ADRBASE_CMD_EXTRA: UINT := ADRBASE_CMD_WARN + COUNT_WARN * 4;
	ADRBASE_CMD_DEVICE: UINT := ADRBASE_CMD_EXTRA + COUNT_EXTRA_CMD;
	
(*	|25001 - 30000| - Резерв *)
(*	|30001 - 35000| - C_SE_NB_1
		sys_logic_nb
		sys_valve.start				x COUNT_VALVE
				 .moving
				 .press
		sys_unit.switch				x COUNT_UNIT
				.work
		device NB
*)
	ADRBASE_NB_LOGIC: UINT := 0;//ADRBASE_IEC_C_SE_NB_1;
	ADRBASE_NB_VALVE: UINT := ADRBASE_NB_LOGIC + COUNT_SP_NB;
	ADRBASE_NB_UNIT: UINT := ADRBASE_NB_VALVE + COUNT_VALVE * 3;
	ADRBASE_NB_EXTRA: UINT := ADRBASE_NB_UNIT + COUNT_UNIT * 2;
	ADRBASE_NB_DEVICE: UINT := ADRBASE_NB_EXTRA + COUNT_EXTRA_NB;
	
(*	|35001 - 40000| - C_SE_NC_1
		sys_logic_nc
		sys_ai.out_min				x COUNT_AI
			  .out_max
			  .delta
			  .val_fail_min
			  .val_fail_max
			  .val_warn_min
			  .val_warn_max
			  .hyst
		sys_ao.tr					x COUNT_AO
			  .in_min
			  .in_max
		device NC
*)		
	ADRBASE_NC_LOGIC: UINT := 0;//ADRBASE_IEC_C_SE_NC_1;
	ADRBASE_NC_TI: UINT := ADRBASE_NC_LOGIC + COUNT_SP_NC;
	ADRBASE_NC_TR: UINT := ADRBASE_NC_TI + MAX_COUNT_AI * 8;
	ADRBASE_NC_EXTRA: UINT := ADRBASE_NC_TR + MAX_COUNT_AO * 3;
	ADRBASE_NC_DEVICE: UINT := ADRBASE_NC_EXTRA + COUNT_EXTRA_NC;
	
(*	|40001 - 65535| - Резерв *)
	
END_VAR

// A1_01A/Application/DEV
VAR_GLOBAL
	// Modbus protocol
	modbus_ip: ARRAY[0.._S_COUNT_PORT_ETH] OF RLTM.RTUMaster;
	modbus_rs: ARRAY[0.._S_COUNT_PORT_SERIAL] OF RLTM.RTUMaster;
	
	//Устройства
	skp: SKP;
	akp: AKP;
	ngk_ipkz_xn: NGK_IPKZ;
	vopetm: VOPETM;
	mercury: Mercury;
	ek: EK;
	testGRS: TestGRS; 
	eris:ERIS;
END_VAR

// Exchange/IP_Message_const
VAR_GLOBAL CONSTANT
	MSG_SIZE : UINT := 8192;

END_VAR

// Serial_port/SerialConst
{attribute 'qualified_only'}
VAR_GLOBAL CONSTANT
	
	START_BYTE		: BYTE := 16#0A;
	
	HALF_MASTER		: UINT := 1;
	HALF_SLAVE		: UINT := 2;
	FULL			: UINT := 3;
	
END_VAR

// IP_Const
VAR_GLOBAL CONSTANT
	SERVER_MAX_CONNECTIONS	: UINT := 32;
	SERVER_MAX_COUNT		: UINT := 16;
	SERVER_TTL_TIME			: TIME := T#5M;
	CLIENT_TTL_TIME			: TIME := T#2M;
	
	CLIENT_MAX_COUNT		: UINT := 16;
	
	WORK_CONNECTION			: UINT := 0;
	OPEN_CONNECTION			: UINT := 1;
	CLOSE_CONNECTION		: UINT := 2;
	REOPEN_CONNECTION		: UINT := 3;	

END_VAR

// A1_01A/Application/Main
PROGRAM Main
VAR
	step: UINT;
	i : UINT;
	bc: BOOL;
END_VAR


CASE (step) OF
	0:
		Init_Gen();
		Init_Main();
		Init_User();
		
		App104.srv.port := sys_server[0].port;
		App104.srv.commonASDUAddress := sys_server[0].asdu;
		App104.srv.windowSizeK := sys_server[0].k;
		App104.srv.windowSizeW := sys_server[0].w;
		App104.srv.timeoutK := UDINT_TO_TIME(UINT_TO_UDINT(sys_server[0].t3) * 1000);
		
		App104.enable := 1;
		Devices.enable := 1;
		step := step + 1;
		
	
	1:
		Cyclic_In();
		Cyclic_Main();
		
		Cyclic_Station();
		
		Cyclic_User();
		
		Cyclic_Out();
		
		bc := FALSE;
		i := 0; WHILE i < COUNT_DO DO
			sys_do[i].cmd_off := NOT sys_do[i].cmd_on;
			sys_do[i]();
			bc := bc OR sys_do[i].sb;
			i := i + 1;
		END_WHILE
		station.global_imit_do := bc;
		
		bc := FALSE;
		i := 0; WHILE i < COUNT_AO DO
			sys_ao_sp[i*3+0]();
			sys_ao_sp[i*3+1]();
			sys_ao_sp[i*3+2]();
			
			sys_ao[i].tr := sys_ao_sp[i*3+0].sp.re;
			sys_ao[i].in_min := sys_ao_sp[i*3+1].sp.re;
			sys_ao[i].in_max := sys_ao_sp[i*3+2].sp.re;
			
			sys_ao[i]();
			bc := bc OR sys_ao[i].sb;
			i := i + 1;
		END_WHILE
		station.global_imit_ao := bc;
		
		Cyclic_DB();
END_CASE

METHOD Init_Main
VAR_INPUT
END_VAR
VAR
	i, N: UINT;
END_VAR
Init_Gen();
Cyclic_In();

fram.count_byte := COUNT_VALVE + COUNT_STOP + COUNT_UNIT + COUNT_FAIL + COUNT_WARN + COUNT_FREESP_BYTE;	// block, block, block, mask, mask, free
fram.count_word := COUNT_VALVE*3 + COUNT_UNIT*2 + COUNT_FREESP_WORD;	// (start, move, press), (switch, work), free		+COUNT_STOP wait time?
fram.count_dword := COUNT_AI*8 + COUNT_AO*3 + COUNT_FREESP_DWORD;	// (s_min, s_max, delta, f_min, f_max, w_min, w_max, hyst), (value, s_min, s_max), free
fram.Init();

i := 0; WHILE i < COUNT_DI DO
	sys_di[i]();
	i := i + 1;
END_WHILE

//count_byte
N := 0;
i := 0; WHILE i < COUNT_VALVE DO
	sys_valve_m[i].pfram := ADR(fram);
	sys_valve_m[i].sp_type := RLTBIO.fram_type.fram_byte;
	sys_valve_m[i].id := N + i;
	sys_valve_m[i].spi.b := FALSE;
	sys_valve_m[i]();
	IF sys_valve_m[i].sp.b THEN
		sys_valve[i].cmd.block_on := TRUE;
	END_IF
	sys_valve[i]();
	i := i + 1;
END_WHILE
N := COUNT_VALVE;
i := 0; WHILE i < COUNT_STOP DO
	sys_stop_m[i].pfram := ADR(fram);
	sys_stop_m[i].sp_type := RLTBIO.fram_type.fram_byte;
	sys_stop_m[i].id := N + i;
	sys_stop_m[i].spi.b := FALSE;
	sys_stop_m[i]();
	
	sys_stop[i].ptr.valve_actions := ADR(sys_stop_actions[i]);
	sys_stop[i].ptr.stops := ADR(sys_stop);
	sys_stop[i].ptr.valves := ADR(sys_valve);
	sys_stop[i].ptr.units := ADR(sys_unit);
	//sys_stop[i].ptr.station := ADR(station);
	sys_stop[i].valve_count := COUNT_VALVE;
	sys_stop[i].unit_count := COUNT_UNIT;
	sys_stop[i].stop_count := COUNT_STOP;
	IF sys_stop_m[i].sp.b THEN
		sys_stop[i].cmd.block_on := TRUE;
	END_IF
	sys_stop[i]();
	i := i + 1;
END_WHILE
N := COUNT_VALVE + COUNT_STOP;
i := 0; WHILE i < COUNT_UNIT DO
	sys_unit_m[i].pfram := ADR(fram);
	sys_unit_m[i].sp_type := RLTBIO.fram_type.fram_byte;
	sys_unit_m[i].id := N + i;
	sys_unit_m[i].spi.b := FALSE;
	sys_unit_m[i]();
	IF sys_unit_m[i].sp.b THEN
		sys_unit[i].cmd.block_on := TRUE;
	END_IF
	sys_unit[i]();
	i := i + 1;
END_WHILE
N := COUNT_VALVE + COUNT_STOP + COUNT_UNIT;
i := 0; WHILE i < COUNT_FAIL DO
	sys_fail_m[i].pfram := ADR(fram);
	sys_fail_m[i].sp_type := RLTBIO.fram_type.fram_byte;
	sys_fail_m[i].id := N + i;
	sys_fail_m[i].spi.b := FALSE;
	sys_fail_m[i]();
	sys_fail[i].block := sys_fail_m[i].sp.b;
	sys_fail[i].type_ack := 1;
	i := i + 1;
END_WHILE
N := COUNT_VALVE + COUNT_STOP + COUNT_UNIT + COUNT_FAIL;
i := 0; WHILE i < COUNT_WARN DO
	sys_warn_m[i].pfram := ADR(fram);
	sys_warn_m[i].sp_type := RLTBIO.fram_type.fram_byte;
	sys_warn_m[i].id := N + i;
	sys_warn_m[i].spi.b := FALSE;
	sys_warn_m[i]();
	sys_warn[i].block := sys_warn_m[i].sp.b;
	i := i + 1;
END_WHILE
(*	копия вынесена в  для возможности задания начальных значений. если это не надо, удалить оттуда и раскомментировать
N := COUNT_VALVE + COUNT_STOP + COUNT_UNIT + COUNT_FAIL + COUNT_WARN;
i := 0; WHILE i < COUNT_FREESP_BYTE DO
	sys_sp_byte[i].pfram := ADR(fram);
	sys_sp_byte[i].sp_type := RLTBIO.fram_type.fram_byte;
	sys_sp_byte[i].id := N + i;
	sys_sp_byte[i].spi.b := FALSE;
	sys_sp_byte[i]();
	i := i + 1;
END_WHILE *)


//count_word
N := 0;
i := 0; WHILE i < COUNT_VALVE DO
	sys_valve_sp[i*3+0].pfram := ADR(fram);
	sys_valve_sp[i*3+0].sp_type := RLTBIO.fram_type.fram_word;
	sys_valve_sp[i*3+0].id := N + i*3+0;
	// spi.ui is @ Init_Gen
	sys_valve_sp[i*3+0]();
	sys_valve_sp[i*3+1].pfram := ADR(fram);
	sys_valve_sp[i*3+1].sp_type := RLTBIO.fram_type.fram_word;
	sys_valve_sp[i*3+1].id := N + i*3+1;
	sys_valve_sp[i*3+1]();
	sys_valve_sp[i*3+2].pfram := ADR(fram);
	sys_valve_sp[i*3+2].sp_type := RLTBIO.fram_type.fram_word;
	sys_valve_sp[i*3+2].id := N + i*3+2;
	sys_valve_sp[i*3+2]();
	
	sys_valve[i].sp.cvw := 3;
	sys_valve[i].sp.start := sys_valve_sp[i*3+0].sp.ui;
	sys_valve[i].sp.moving := sys_valve_sp[i*3+1].sp.ui;
	sys_valve[i].sp.press := sys_valve_sp[i*3+2].sp.ui;
	sys_valve[i].sp.imit := 3;
	sys_valve[i].sp.sol := 1;
	
	sys_valve[i]();
	i := i + 1;
END_WHILE
N := COUNT_VALVE*3;
i := 0; WHILE i < COUNT_UNIT DO
	sys_unit_sp[i*2+0].pfram := ADR(fram);
	sys_unit_sp[i*2+0].sp_type := RLTBIO.fram_type.fram_word;
	sys_unit_sp[i*2+0].id := N + i*2+0;
	// spi.ui is @ Init_Gen
	sys_unit_sp[i*2+0]();
	sys_unit_sp[i*2+1].pfram := ADR(fram);
	sys_unit_sp[i*2+1].sp_type := RLTBIO.fram_type.fram_word;
	sys_unit_sp[i*2+1].id := N + i*2+1;
	sys_unit_sp[i*2+1]();
	
	sys_unit[i].sp.cvw := 3;
	sys_unit[i].sp.switch := sys_unit_sp[i*2+0].sp.ui;
	sys_unit[i].sp.work := sys_unit_sp[i*2+1].sp.ui;
	sys_unit[i].sp.imit := 1;
	
	sys_unit[i]();
	i := i + 1;
END_WHILE
(*	копия вынесена в  для возможности задания начальных значений. если это не надо, удалить оттуда и раскомментировать
N := COUNT_VALVE*3 + COUNT_UNIT*2;
i := 0; WHILE i < COUNT_FREESP_WORD DO
	sys_sp_word[i].pfram := ADR(fram);
	sys_sp_word[i].sp_type := RLTBIO.fram_type.fram_word;
	sys_sp_word[i].id := N + i;
	sys_sp_word[i].spi.ui := 0;
	sys_sp_word[i]();
	i := i + 1;
END_WHILE	*)


//count_dword
N := 0;
i := 0; WHILE i < COUNT_AI DO
	sys_ai_sp[i*8+0].pfram := ADR(fram);
	sys_ai_sp[i*8+0].sp_type := RLTBIO.fram_type.fram_dword;
	sys_ai_sp[i*8+0].id := N + i*8+0;
	// spi.re is @ Init_Gen
	sys_ai_sp[i*8+0]();
	sys_ai_sp[i*8+1].pfram := ADR(fram);
	sys_ai_sp[i*8+1].sp_type := RLTBIO.fram_type.fram_dword;
	sys_ai_sp[i*8+1].id := N + i*8+1;
	sys_ai_sp[i*8+1]();
	sys_ai_sp[i*8+2].pfram := ADR(fram);
	sys_ai_sp[i*8+2].sp_type := RLTBIO.fram_type.fram_dword;
	sys_ai_sp[i*8+2].id := N + i*8+2;
	sys_ai_sp[i*8+2]();
	sys_ai_sp[i*8+3].pfram := ADR(fram);
	sys_ai_sp[i*8+3].sp_type := RLTBIO.fram_type.fram_dword;
	sys_ai_sp[i*8+3].id := N + i*8+3;
	sys_ai_sp[i*8+3]();
	sys_ai_sp[i*8+4].pfram := ADR(fram);
	sys_ai_sp[i*8+4].sp_type := RLTBIO.fram_type.fram_dword;
	sys_ai_sp[i*8+4].id := N + i*8+4;
	sys_ai_sp[i*8+4]();
	sys_ai_sp[i*8+5].pfram := ADR(fram);
	sys_ai_sp[i*8+5].sp_type := RLTBIO.fram_type.fram_dword;
	sys_ai_sp[i*8+5].id := N + i*8+5;
	sys_ai_sp[i*8+5]();
	sys_ai_sp[i*8+6].pfram := ADR(fram);
	sys_ai_sp[i*8+6].sp_type := RLTBIO.fram_type.fram_dword;
	sys_ai_sp[i*8+6].id := N + i*8+6;
	sys_ai_sp[i*8+6]();
	sys_ai_sp[i*8+7].pfram := ADR(fram);
	sys_ai_sp[i*8+7].sp_type := RLTBIO.fram_type.fram_dword;
	sys_ai_sp[i*8+7].id := N + i*8+7;
	sys_ai_sp[i*8+7]();
	
	sys_ai[i].out_min := sys_ai_sp[i*8+0].sp.re;
	sys_ai[i].out_max := sys_ai_sp[i*8+1].sp.re;
	sys_ai[i].delta := sys_ai_sp[i*8+2].sp.re;
	sys_ai[i].val_fail_min := sys_ai_sp[i*8+3].sp.re;
	sys_ai[i].val_fail_max := sys_ai_sp[i*8+4].sp.re;
	sys_ai[i].val_warn_min := sys_ai_sp[i*8+5].sp.re;
	sys_ai[i].val_warn_max := sys_ai_sp[i*8+6].sp.re;
	sys_ai[i].hyst := sys_ai_sp[i*8+7].sp.re;
	
	sys_ai[i]();
	i := i + 1;
END_WHILE
N := COUNT_AI*8;
i := 0; WHILE i < COUNT_AO DO
	sys_ao_sp[i*3+0].pfram := ADR(fram);
	sys_ao_sp[i*3+0].sp_type := RLTBIO.fram_type.fram_dword;
	sys_ao_sp[i*3+0].id := N + i*3+0;
	// spi.re is @ Init_Gen
	sys_ao_sp[i*3+0]();
	sys_ao_sp[i*3+1].pfram := ADR(fram);
	sys_ao_sp[i*3+1].sp_type := RLTBIO.fram_type.fram_dword;
	sys_ao_sp[i*3+1].id := N + i*3+1;
	sys_ao_sp[i*3+1]();
	sys_ao_sp[i*3+2].pfram := ADR(fram);
	sys_ao_sp[i*3+2].sp_type := RLTBIO.fram_type.fram_dword;
	sys_ao_sp[i*3+2].id := N + i*3+2;
	sys_ao_sp[i*3+2]();
	
	sys_ao[i].tr := sys_ao_sp[i*3+0].sp.re;
	sys_ao[i].in_min := sys_ao_sp[i*3+1].sp.re;
	sys_ao[i].in_max := sys_ao_sp[i*3+2].sp.re;
	
	sys_ao[i]();
	i := i + 1;
END_WHILE
(*	копия вынесена в  для возможности задания начальных значений. если это не надо, удалить оттуда и раскомментировать
N := COUNT_AI*8 + COUNT_AO*3;
i := 0; WHILE i < COUNT_FREESP_DWORD DO
	sys_sp_dword[i].pfram := ADR(fram);
	sys_sp_dword[i].sp_type := RLTBIO.fram_type.fram_dword;
	sys_sp_dword[i].id := N + i;
	sys_sp_dword[i].spi.re := 0.0;
	sys_sp_dword[i]();
	i := i + 1;
END_WHILE	*)


i := 0; WHILE i < MIN(COUNT_SERVERS, COUNT_MAX_SERVERS) DO
	station.originators[i] := sys_server[i].originator;
	i := i + 1;
END_WHILE
station.originators[0] := 0;	// SELF always 0

IF station.num_di_valve_dist >= CFG.COUNT_DI THEN
	station.num_di_valve_dist := CFG.COUNT_DI;
	station.cfg.conf_valve_dist := FALSE;
	station.err_num := TRUE;
END_IF
//IF station.num_di_valve_cv >= CFG.COUNT_DI THEN
//	station.num_di_valve_cv := CFG.COUNT_DI;
//	station.cfg.conf_valve_cv := FALSE;
//	station.err_num := TRUE;
//END_IF
IF station.num_do_valve_cv >= CFG.COUNT_DO THEN
	station.num_do_valve_cv := CFG.COUNT_DO;
	station.cfg.conf_valve_cv := FALSE;
	station.err_num := TRUE;
END_IF
IF station.num_di_unit_dist >= CFG.COUNT_DI THEN
	station.num_di_unit_dist := CFG.COUNT_DI;
	station.cfg.conf_unit_dist := FALSE;
	station.err_num := TRUE;
END_IF
//IF station.num_di_unit_cv >= CFG.COUNT_DI THEN
//	station.num_di_unit_cv := CFG.COUNT_DI;
//	station.cfg.conf_unit_cv := FALSE;
//	station.err_num := TRUE;
//END_IF
IF station.num_do_unit_cv >= CFG.COUNT_DO THEN
	station.num_do_unit_cv := CFG.COUNT_DO;
	station.cfg.conf_unit_cv := FALSE;
	station.err_num := TRUE;
END_IF

IF station.num_di_stop_1 >= CFG.COUNT_DI THEN
	station.num_di_stop_1 := CFG.COUNT_DI;
	station.cfg.conf_stop_1 := FALSE;
	station.err_num := TRUE;
END_IF
IF station.num_di_stop_2 >= CFG.COUNT_DI THEN
	station.num_di_stop_2 := CFG.COUNT_DI;
	station.cfg.conf_stop_2 := FALSE;
	station.err_num := TRUE;
END_IF
IF station.num_stop_1 >= CFG.COUNT_STOP THEN
	station.num_stop_1 := CFG.COUNT_STOP;
	station.cfg.conf_stop_1 := FALSE;
	station.err_num := TRUE;
END_IF
IF station.num_stop_2 >= CFG.COUNT_STOP THEN
	station.num_stop_2 := CFG.COUNT_STOP;
	station.cfg.conf_stop_2 := FALSE;
	station.err_num := TRUE;
END_IF

IF station.num_do_sound >= CFG.COUNT_DO THEN
	station.num_do_sound := CFG.COUNT_DO;
	station.cfg.conf_sound := FALSE;
	station.err_num := TRUE;
END_IF
IF station.num_do_alarm >= CFG.COUNT_DO THEN
	station.num_do_alarm := CFG.COUNT_DO;
	station.cfg.conf_alarm := FALSE;
	station.err_num := TRUE;
END_IF
IF station.num_do_lamp_fail >= CFG.COUNT_DO THEN
	station.num_do_lamp_fail := CFG.COUNT_DO;
	station.cfg.conf_fail := FALSE;
	station.err_num := TRUE;
END_IF
IF station.num_do_lamp_alarm >= CFG.COUNT_DO THEN
	station.num_do_lamp_alarm := CFG.COUNT_DO;
	station.cfg.conf_warn := FALSE;
	station.err_num := TRUE;
END_IF
IF station.num_do_lamp_fire >= CFG.COUNT_DO THEN
	station.num_do_lamp_fire := CFG.COUNT_DO;
	station.cfg.conf_fire := FALSE;
	station.err_num := TRUE;
END_IF
IF station.num_do_lamp_gas >= CFG.COUNT_DO THEN
	station.num_do_lamp_gas := CFG.COUNT_DO;
	station.cfg.conf_gas := FALSE;
	station.err_num := TRUE;
END_IF

IF station.num_di_ack >= CFG.COUNT_DI THEN
	station.num_di_ack := CFG.COUNT_DI;
	station.cfg.conf_ack := FALSE;
	station.err_num := TRUE;
END_IF
IF station.num_di_sound >= CFG.COUNT_DI THEN
	station.num_di_sound := CFG.COUNT_DI;
	station.cfg.conf_test_sound := FALSE;
	station.err_num := TRUE;
END_IF
IF station.num_di_alarm >= CFG.COUNT_DI THEN
	station.num_di_alarm := CFG.COUNT_DI;
	station.cfg.conf_test_alarm := FALSE;
	station.err_num := TRUE;
END_IF
IF station.num_di_lamps >= CFG.COUNT_DI THEN
	station.num_di_lamps := CFG.COUNT_DI;
	station.cfg.conf_lamps := FALSE;
	station.err_num := TRUE;
END_IF
END_METHOD

METHOD Init_Gen
VAR_INPUT
END_VAR
    
    StrCpyW(ADR(sys_server[0].name), SIZEOF(sys_server[0].name), ADR("Local"));
    StrCpyW(ADR(sys_server[0].name), SIZEOF(sys_server[0].name), ADR("Self"));
    sys_server[0].originator := 0;
    sys_server[0].asdu := 1;
    sys_server[0].T1 := 15;
    sys_server[0].T2 := 10;
    sys_server[0].T3 := 30;
    sys_server[0].k := 1;
    sys_server[0].w := 1;
    sys_server[0].port := 2404;
    StrCpyW(ADR(sys_server[1].name), SIZEOF(sys_server[1].name), ADR("Main"));
    StrCpyW(ADR(sys_server[1].name), SIZEOF(sys_server[1].name), ADR("Channel#1"));
    sys_server[1].originator := 1;
    sys_server[1].asdu := 1;
    sys_server[1].T1 := 15;
    sys_server[1].T2 := 10;
    sys_server[1].T3 := 30;
    sys_server[1].k := 1;
    sys_server[1].w := 1;
    sys_server[1].port := 2404;
    StrCpyW(ADR(sys_server[2].name), SIZEOF(sys_server[2].name), ADR("Backup"));
    StrCpyW(ADR(sys_server[2].name), SIZEOF(sys_server[2].name), ADR("Channel#1"));
    sys_server[2].originator := 2;
    sys_server[2].asdu := 1;
    sys_server[2].T1 := 15;
    sys_server[2].T2 := 10;
    sys_server[2].T3 := 30;
    sys_server[2].k := 1;
    sys_server[2].w := 1;
    sys_server[2].port := 2404;
    StrCpyW(ADR(sys_server[3].name), SIZEOF(sys_server[3].name), ADR("Service"));
    StrCpyW(ADR(sys_server[3].name), SIZEOF(sys_server[3].name), ADR("Channel#1"));
    sys_server[3].originator := 3;
    sys_server[3].asdu := 1;
    sys_server[3].T1 := 15;
    sys_server[3].T2 := 10;
    sys_server[3].T3 := 30;
    sys_server[3].k := 1;
    sys_server[3].w := 1;
    sys_server[3].port := 2404;
    
    StrCpyW(ADR(sys_mod[0].name), SIZEOF(sys_mod[0].name), ADR("ПР"));
    sys_mod[0].id := 0;
    StrCpyW(ADR(sys_mod[1].name), SIZEOF(sys_mod[1].name), ADR("ВДС-32"));
    sys_mod[1].id := 1;
    StrCpyW(ADR(sys_mod[2].name), SIZEOF(sys_mod[2].name), ADR("ВДС-16/ВТУ-16"));
    sys_mod[2].id := 2;
    StrCpyW(ADR(sys_mod[3].name), SIZEOF(sys_mod[3].name), ADR("ВТИ-16"));
    sys_mod[3].id := 3;
    
    //StrCpyW(ADR(sys_di[0].name), SIZEOF(sys_di[0].name), ADR("Кран № 388.7 открыт"));
    sys_di[0].fail := FALSE;
    sys_di[0].klv := 2;
    sys_di[0].m := 3;
    sys_di[0].t0 := UDINT_TO_TIME(10);
    sys_di[0].inv := 0;
    //StrCpyW(ADR(sys_di[1].name), SIZEOF(sys_di[1].name), ADR("Кран № 388.7 закрыт"));
    sys_di[1].fail := FALSE;
    sys_di[1].klv := 2;
    sys_di[1].m := 3;
    sys_di[1].t0 := UDINT_TO_TIME(10);
    sys_di[1].inv := 0;
    //StrCpyW(ADR(sys_di[2].name), SIZEOF(sys_di[2].name), ADR("Контроль цепей Крана № 388.7 соленоид открытия"));
    sys_di[2].fail := FALSE;
    sys_di[2].klv := 2;
    sys_di[2].m := 3;
    sys_di[2].t0 := UDINT_TO_TIME(10);
    sys_di[2].inv := 0;
    //StrCpyW(ADR(sys_di[3].name), SIZEOF(sys_di[3].name), ADR("Контроль цепей Крана № 388.7 соленоид закрытия"));
    sys_di[3].fail := FALSE;
    sys_di[3].klv := 2;
    sys_di[3].m := 3;
    sys_di[3].t0 := UDINT_TO_TIME(10);
    sys_di[3].inv := 0;
    //StrCpyW(ADR(sys_di[4].name), SIZEOF(sys_di[4].name), ADR("Кран № 2 открыт (Резерв)"));
    sys_di[4].fail := FALSE;
    sys_di[4].klv := 2;
    sys_di[4].m := 3;
    sys_di[4].t0 := UDINT_TO_TIME(10);
    sys_di[4].inv := 0;
    //StrCpyW(ADR(sys_di[5].name), SIZEOF(sys_di[5].name), ADR("Кран № 2 закрыт (Резерв)"));
    sys_di[5].fail := FALSE;
    sys_di[5].klv := 2;
    sys_di[5].m := 3;
    sys_di[5].t0 := UDINT_TO_TIME(10);
    sys_di[5].inv := 0;
    //StrCpyW(ADR(sys_di[6].name), SIZEOF(sys_di[6].name), ADR("Контроль цепей крана 2 соленоид открытия (Резерв)"));
    sys_di[6].fail := FALSE;
    sys_di[6].klv := 2;
    sys_di[6].m := 3;
    sys_di[6].t0 := UDINT_TO_TIME(10);
    sys_di[6].inv := 0;
    //StrCpyW(ADR(sys_di[7].name), SIZEOF(sys_di[7].name), ADR("Контроль цепей крана 2 соленоид закрытия (Резерв)"));
    sys_di[7].fail := FALSE;
    sys_di[7].klv := 2;
    sys_di[7].m := 3;
    sys_di[7].t0 := UDINT_TO_TIME(10);
    sys_di[7].inv := 0;
    //StrCpyW(ADR(sys_di[8].name), SIZEOF(sys_di[8].name), ADR("Шкаф КП ТМ открыт (инверсный)"));
    sys_di[8].fail := FALSE;
    sys_di[8].klv := 2;
    sys_di[8].m := 3;
    sys_di[8].t0 := UDINT_TO_TIME(10);
    sys_di[8].inv := 0;
    //StrCpyW(ADR(sys_di[9].name), SIZEOF(sys_di[9].name), ADR("ТС Блок питания кранов (=24В/24В) в норме"));
    sys_di[9].fail := FALSE;
    sys_di[9].klv := 2;
    sys_di[9].m := 3;
    sys_di[9].t0 := UDINT_TO_TIME(10);
    sys_di[9].inv := 0;
    //StrCpyW(ADR(sys_di[10].name), SIZEOF(sys_di[10].name), ADR("Контроль изоляции цепей питания кранов (инверсный)"));
    sys_di[10].fail := FALSE;
    sys_di[10].klv := 2;
    sys_di[10].m := 3;
    sys_di[10].t0 := UDINT_TO_TIME(10);
    sys_di[10].inv := 0;
    //StrCpyW(ADR(sys_di[11].name), SIZEOF(sys_di[11].name), ADR("Контроль изоляции цепей питания внутри шкафа (инверсный)"));
    sys_di[11].fail := FALSE;
    sys_di[11].klv := 2;
    sys_di[11].m := 3;
    sys_di[11].t0 := UDINT_TO_TIME(10);
    sys_di[11].inv := 0;
    //StrCpyW(ADR(sys_di[12].name), SIZEOF(sys_di[12].name), ADR("Подготовка ТУ"));
    sys_di[12].fail := FALSE;
    sys_di[12].klv := 2;
    sys_di[12].m := 3;
    sys_di[12].t0 := UDINT_TO_TIME(10);
    sys_di[12].inv := 0;
    //StrCpyW(ADR(sys_di[13].name), SIZEOF(sys_di[13].name), ADR("Режим управления дистанционный"));
    sys_di[13].fail := FALSE;
    sys_di[13].klv := 2;
    sys_di[13].m := 3;
    sys_di[13].t0 := UDINT_TO_TIME(10);
    sys_di[13].inv := 0;
    //StrCpyW(ADR(sys_di[14].name), SIZEOF(sys_di[14].name), ADR("Режим проверки ламп"));
    sys_di[14].fail := FALSE;
    sys_di[14].klv := 2;
    sys_di[14].m := 3;
    sys_di[14].t0 := UDINT_TO_TIME(10);
    sys_di[14].inv := 0;
    //StrCpyW(ADR(sys_di[15].name), SIZEOF(sys_di[15].name), ADR("Резерв"));
    sys_di[15].fail := FALSE;
    sys_di[15].klv := 2;
    sys_di[15].m := 3;
    sys_di[15].t0 := UDINT_TO_TIME(10);
    sys_di[15].inv := 0;
    //StrCpyW(ADR(sys_di[16].name), SIZEOF(sys_di[16].name), ADR("ИБП. Шкаф открыт (инверсный)"));
    sys_di[16].fail := FALSE;
    sys_di[16].klv := 2;
    sys_di[16].m := 3;
    sys_di[16].t0 := UDINT_TO_TIME(10);
    sys_di[16].inv := 0;
    //StrCpyW(ADR(sys_di[17].name), SIZEOF(sys_di[17].name), ADR("ИБП. Работает система микроклимата (инверсный)"));
    sys_di[17].fail := FALSE;
    sys_di[17].klv := 2;
    sys_di[17].m := 3;
    sys_di[17].t0 := UDINT_TO_TIME(10);
    sys_di[17].inv := 0;
    //StrCpyW(ADR(sys_di[18].name), SIZEOF(sys_di[18].name), ADR("ИБП. Сработал автоматический выключатель"));
    sys_di[18].fail := FALSE;
    sys_di[18].klv := 2;
    sys_di[18].m := 3;
    sys_di[18].t0 := UDINT_TO_TIME(10);
    sys_di[18].inv := 0;
    //StrCpyW(ADR(sys_di[19].name), SIZEOF(sys_di[19].name), ADR("ИБП. Наличие сетевого напряжения 220В"));
    sys_di[19].fail := FALSE;
    sys_di[19].klv := 2;
    sys_di[19].m := 3;
    sys_di[19].t0 := UDINT_TO_TIME(10);
    sys_di[19].inv := 0;
    //StrCpyW(ADR(sys_di[20].name), SIZEOF(sys_di[20].name), ADR("ИБП. Напряжение на АКБ ниже 20,5В"));
    sys_di[20].fail := FALSE;
    sys_di[20].klv := 2;
    sys_di[20].m := 3;
    sys_di[20].t0 := UDINT_TO_TIME(10);
    sys_di[20].inv := 0;
    //StrCpyW(ADR(sys_di[21].name), SIZEOF(sys_di[21].name), ADR("ИБП. Работает от АКБ"));
    sys_di[21].fail := FALSE;
    sys_di[21].klv := 2;
    sys_di[21].m := 3;
    sys_di[21].t0 := UDINT_TO_TIME(10);
    sys_di[21].inv := 0;
    //StrCpyW(ADR(sys_di[22].name), SIZEOF(sys_di[22].name), ADR("Резерв"));
    sys_di[22].fail := FALSE;
    sys_di[22].klv := 2;
    sys_di[22].m := 3;
    sys_di[22].t0 := UDINT_TO_TIME(10);
    sys_di[22].inv := 0;
    //StrCpyW(ADR(sys_di[23].name), SIZEOF(sys_di[23].name), ADR("ИБП. Защита по входу 220В исправна (резерв)"));
    sys_di[23].fail := FALSE;
    sys_di[23].klv := 2;
    sys_di[23].m := 3;
    sys_di[23].t0 := UDINT_TO_TIME(10);
    sys_di[23].inv := 0;
    //StrCpyW(ADR(sys_di[24].name), SIZEOF(sys_di[24].name), ADR("БКЭС. Активная энергия на вводе 0,4 кВ"));
    sys_di[24].fail := FALSE;
    sys_di[24].klv := 2;
    sys_di[24].m := 3;
    sys_di[24].t0 := UDINT_TO_TIME(10);
    sys_di[24].inv := 0;
    //StrCpyW(ADR(sys_di[25].name), SIZEOF(sys_di[25].name), ADR("БКЭС. Тревога в блок-боксе БКЭС"));
    sys_di[25].fail := FALSE;
    sys_di[25].klv := 2;
    sys_di[25].m := 3;
    sys_di[25].t0 := UDINT_TO_TIME(10);
    sys_di[25].inv := 0;
    //StrCpyW(ADR(sys_di[26].name), SIZEOF(sys_di[26].name), ADR("БКЭС. Наличие напряжения на вводе 0,4 кВ"));
    sys_di[26].fail := FALSE;
    sys_di[26].klv := 2;
    sys_di[26].m := 3;
    sys_di[26].t0 := UDINT_TO_TIME(10);
    sys_di[26].inv := 0;
    //StrCpyW(ADR(sys_di[27].name), SIZEOF(sys_di[27].name), ADR("БКЭС. Включен QF1"));
    sys_di[27].fail := FALSE;
    sys_di[27].klv := 2;
    sys_di[27].m := 3;
    sys_di[27].t0 := UDINT_TO_TIME(10);
    sys_di[27].inv := 0;
    //StrCpyW(ADR(sys_di[28].name), SIZEOF(sys_di[28].name), ADR("БКЭС. Неисправность  АУПС"));
    sys_di[28].fail := FALSE;
    sys_di[28].klv := 2;
    sys_di[28].m := 3;
    sys_di[28].t0 := UDINT_TO_TIME(10);
    sys_di[28].inv := 0;
    //StrCpyW(ADR(sys_di[29].name), SIZEOF(sys_di[29].name), ADR("БКЭС. Пожар в блок-боксе БКЭС"));
    sys_di[29].fail := FALSE;
    sys_di[29].klv := 2;
    sys_di[29].m := 3;
    sys_di[29].t0 := UDINT_TO_TIME(10);
    sys_di[29].inv := 0;
    //StrCpyW(ADR(sys_di[30].name), SIZEOF(sys_di[30].name), ADR("БКЭС. Выключатель нагрузки QS1 включен"));
    sys_di[30].fail := FALSE;
    sys_di[30].klv := 2;
    sys_di[30].m := 3;
    sys_di[30].t0 := UDINT_TO_TIME(10);
    sys_di[30].inv := 0;
    //StrCpyW(ADR(sys_di[31].name), SIZEOF(sys_di[31].name), ADR("БКЭС. Заземляющий нож выключатель нагрузки QS1 включен"));
    sys_di[31].fail := FALSE;
    sys_di[31].klv := 2;
    sys_di[31].m := 3;
    sys_di[31].t0 := UDINT_TO_TIME(10);
    sys_di[31].inv := 0;
    //StrCpyW(ADR(sys_di[32].name), SIZEOF(sys_di[32].name), ADR("Тревога на площадке крана 388.7"));
    sys_di[32].fail := FALSE;
    sys_di[32].klv := 2;
    sys_di[32].m := 3;
    sys_di[32].t0 := UDINT_TO_TIME(10);
    sys_di[32].inv := 0;
    //StrCpyW(ADR(sys_di[33].name), SIZEOF(sys_di[33].name), ADR("Тревога в блок-боксе КП ТМ"));
    sys_di[33].fail := FALSE;
    sys_di[33].klv := 2;
    sys_di[33].m := 3;
    sys_di[33].t0 := UDINT_TO_TIME(10);
    sys_di[33].inv := 0;
    //StrCpyW(ADR(sys_di[34].name), SIZEOF(sys_di[34].name), ADR("Авария источника питания охранной сигнализации"));
    sys_di[34].fail := FALSE;
    sys_di[34].klv := 2;
    sys_di[34].m := 3;
    sys_di[34].t0 := UDINT_TO_TIME(10);
    sys_di[34].inv := 0;
    //StrCpyW(ADR(sys_di[35].name), SIZEOF(sys_di[35].name), ADR("Резерв"));
    sys_di[35].fail := FALSE;
    sys_di[35].klv := 2;
    sys_di[35].m := 3;
    sys_di[35].t0 := UDINT_TO_TIME(10);
    sys_di[35].inv := 0;
    //StrCpyW(ADR(sys_di[36].name), SIZEOF(sys_di[36].name), ADR("Резерв"));
    sys_di[36].fail := FALSE;
    sys_di[36].klv := 2;
    sys_di[36].m := 3;
    sys_di[36].t0 := UDINT_TO_TIME(10);
    sys_di[36].inv := 0;
    //StrCpyW(ADR(sys_di[37].name), SIZEOF(sys_di[37].name), ADR("Резерв"));
    sys_di[37].fail := FALSE;
    sys_di[37].klv := 2;
    sys_di[37].m := 3;
    sys_di[37].t0 := UDINT_TO_TIME(10);
    sys_di[37].inv := 0;
    //StrCpyW(ADR(sys_di[38].name), SIZEOF(sys_di[38].name), ADR("Резерв"));
    sys_di[38].fail := FALSE;
    sys_di[38].klv := 2;
    sys_di[38].m := 3;
    sys_di[38].t0 := UDINT_TO_TIME(10);
    sys_di[38].inv := 0;
    //StrCpyW(ADR(sys_di[39].name), SIZEOF(sys_di[39].name), ADR("Резерв"));
    sys_di[39].fail := FALSE;
    sys_di[39].klv := 2;
    sys_di[39].m := 3;
    sys_di[39].t0 := UDINT_TO_TIME(10);
    sys_di[39].inv := 0;
    //StrCpyW(ADR(sys_di[40].name), SIZEOF(sys_di[40].name), ADR("Резерв"));
    sys_di[40].fail := FALSE;
    sys_di[40].klv := 2;
    sys_di[40].m := 3;
    sys_di[40].t0 := UDINT_TO_TIME(10);
    sys_di[40].inv := 0;
    //StrCpyW(ADR(sys_di[41].name), SIZEOF(sys_di[41].name), ADR("Резерв"));
    sys_di[41].fail := FALSE;
    sys_di[41].klv := 2;
    sys_di[41].m := 3;
    sys_di[41].t0 := UDINT_TO_TIME(10);
    sys_di[41].inv := 0;
    //StrCpyW(ADR(sys_di[42].name), SIZEOF(sys_di[42].name), ADR("Резерв"));
    sys_di[42].fail := FALSE;
    sys_di[42].klv := 2;
    sys_di[42].m := 3;
    sys_di[42].t0 := UDINT_TO_TIME(10);
    sys_di[42].inv := 0;
    //StrCpyW(ADR(sys_di[43].name), SIZEOF(sys_di[43].name), ADR("Резерв"));
    sys_di[43].fail := FALSE;
    sys_di[43].klv := 2;
    sys_di[43].m := 3;
    sys_di[43].t0 := UDINT_TO_TIME(10);
    sys_di[43].inv := 0;
    //StrCpyW(ADR(sys_di[44].name), SIZEOF(sys_di[44].name), ADR("Резерв"));
    sys_di[44].fail := FALSE;
    sys_di[44].klv := 2;
    sys_di[44].m := 3;
    sys_di[44].t0 := UDINT_TO_TIME(10);
    sys_di[44].inv := 0;
    //StrCpyW(ADR(sys_di[45].name), SIZEOF(sys_di[45].name), ADR("Резерв"));
    sys_di[45].fail := FALSE;
    sys_di[45].klv := 2;
    sys_di[45].m := 3;
    sys_di[45].t0 := UDINT_TO_TIME(10);
    sys_di[45].inv := 0;
    //StrCpyW(ADR(sys_di[46].name), SIZEOF(sys_di[46].name), ADR("Резерв"));
    sys_di[46].fail := FALSE;
    sys_di[46].klv := 2;
    sys_di[46].m := 3;
    sys_di[46].t0 := UDINT_TO_TIME(10);
    sys_di[46].inv := 0;
    //StrCpyW(ADR(sys_di[47].name), SIZEOF(sys_di[47].name), ADR("Резерв"));
    sys_di[47].fail := FALSE;
    sys_di[47].klv := 2;
    sys_di[47].m := 3;
    sys_di[47].t0 := UDINT_TO_TIME(10);
    sys_di[47].inv := 0;
    
    //StrCpyW(ADR(sys_do[0].name), SIZEOF(sys_do[0].name), ADR("Кран № 388.7 открыть"));
    sys_do[0].q := 0;
    sys_do[0].t_on := UDINT_TO_TIME(3000);
    sys_do[0].t_off := UDINT_TO_TIME(3000);
    sys_do[0].t_ret := UDINT_TO_TIME(1500);
    //StrCpyW(ADR(sys_do[1].name), SIZEOF(sys_do[1].name), ADR("Кран № 388.7 закрыть"));
    sys_do[1].q := 0;
    sys_do[1].t_on := UDINT_TO_TIME(3000);
    sys_do[1].t_off := UDINT_TO_TIME(3000);
    sys_do[1].t_ret := UDINT_TO_TIME(1500);
    //StrCpyW(ADR(sys_do[2].name), SIZEOF(sys_do[2].name), ADR("Кран № 2 открыть (Резерв)"));
    sys_do[2].q := 0;
    sys_do[2].t_on := UDINT_TO_TIME(3000);
    sys_do[2].t_off := UDINT_TO_TIME(3000);
    sys_do[2].t_ret := UDINT_TO_TIME(1500);
    //StrCpyW(ADR(sys_do[3].name), SIZEOF(sys_do[3].name), ADR("Кран № 2 закрыть (Резерв)"));
    sys_do[3].q := 0;
    sys_do[3].t_on := UDINT_TO_TIME(3000);
    sys_do[3].t_off := UDINT_TO_TIME(3000);
    sys_do[3].t_ret := UDINT_TO_TIME(1500);
    //StrCpyW(ADR(sys_do[4].name), SIZEOF(sys_do[4].name), ADR("Резерв"));
    sys_do[4].q := 0;
    sys_do[4].t_on := UDINT_TO_TIME(3000);
    sys_do[4].t_off := UDINT_TO_TIME(3000);
    sys_do[4].t_ret := UDINT_TO_TIME(1500);
    //StrCpyW(ADR(sys_do[5].name), SIZEOF(sys_do[5].name), ADR("Резерв"));
    sys_do[5].q := 0;
    sys_do[5].t_on := UDINT_TO_TIME(3000);
    sys_do[5].t_off := UDINT_TO_TIME(3000);
    sys_do[5].t_ret := UDINT_TO_TIME(1500);
    //StrCpyW(ADR(sys_do[6].name), SIZEOF(sys_do[6].name), ADR("Резерв"));
    sys_do[6].q := 0;
    sys_do[6].t_on := UDINT_TO_TIME(3000);
    sys_do[6].t_off := UDINT_TO_TIME(3000);
    sys_do[6].t_ret := UDINT_TO_TIME(1500);
    //StrCpyW(ADR(sys_do[7].name), SIZEOF(sys_do[7].name), ADR("Подготовка ТУ"));
    sys_do[7].q := 0;
    sys_do[7].t_on := UDINT_TO_TIME(3000);
    sys_do[7].t_off := UDINT_TO_TIME(3000);
    sys_do[7].t_ret := UDINT_TO_TIME(1500);
    //StrCpyW(ADR(sys_do[8].name), SIZEOF(sys_do[8].name), ADR("Резерв"));
    sys_do[8].q := 0;
    sys_do[8].t_on := UDINT_TO_TIME(3000);
    sys_do[8].t_off := UDINT_TO_TIME(3000);
    sys_do[8].t_ret := UDINT_TO_TIME(1500);
    //StrCpyW(ADR(sys_do[9].name), SIZEOF(sys_do[9].name), ADR("Резерв"));
    sys_do[9].q := 0;
    sys_do[9].t_on := UDINT_TO_TIME(3000);
    sys_do[9].t_off := UDINT_TO_TIME(3000);
    sys_do[9].t_ret := UDINT_TO_TIME(1500);
    //StrCpyW(ADR(sys_do[10].name), SIZEOF(sys_do[10].name), ADR("Резерв"));
    sys_do[10].q := 0;
    sys_do[10].t_on := UDINT_TO_TIME(3000);
    sys_do[10].t_off := UDINT_TO_TIME(3000);
    sys_do[10].t_ret := UDINT_TO_TIME(1500);
    //StrCpyW(ADR(sys_do[11].name), SIZEOF(sys_do[11].name), ADR("Резерв"));
    sys_do[11].q := 0;
    sys_do[11].t_on := UDINT_TO_TIME(3000);
    sys_do[11].t_off := UDINT_TO_TIME(3000);
    sys_do[11].t_ret := UDINT_TO_TIME(1500);
    //StrCpyW(ADR(sys_do[12].name), SIZEOF(sys_do[12].name), ADR("Резерв"));
    sys_do[12].q := 0;
    sys_do[12].t_on := UDINT_TO_TIME(3000);
    sys_do[12].t_off := UDINT_TO_TIME(3000);
    sys_do[12].t_ret := UDINT_TO_TIME(1500);
    //StrCpyW(ADR(sys_do[13].name), SIZEOF(sys_do[13].name), ADR("Резерв"));
    sys_do[13].q := 0;
    sys_do[13].t_on := UDINT_TO_TIME(3000);
    sys_do[13].t_off := UDINT_TO_TIME(3000);
    sys_do[13].t_ret := UDINT_TO_TIME(1500);
    //StrCpyW(ADR(sys_do[14].name), SIZEOF(sys_do[14].name), ADR("Резерв"));
    sys_do[14].q := 0;
    sys_do[14].t_on := UDINT_TO_TIME(3000);
    sys_do[14].t_off := UDINT_TO_TIME(3000);
    sys_do[14].t_ret := UDINT_TO_TIME(1500);
    //StrCpyW(ADR(sys_do[15].name), SIZEOF(sys_do[15].name), ADR("Резерв"));
    sys_do[15].q := 0;
    sys_do[15].t_on := UDINT_TO_TIME(3000);
    sys_do[15].t_off := UDINT_TO_TIME(3000);
    sys_do[15].t_ret := UDINT_TO_TIME(1500);
    
    //StrCpyW(ADR(sys_ai[0].name), SIZEOF(sys_ai[0].name), ADR("Напряжение сетевого питания 220В"));
    //StrCpyW(ADR(sys_ai[0].name), SIZEOF(sys_ai[0].name), ADR("%"));
    sys_ai[0].fail := FALSE;
    sys_ai[0].k := 0.2;
    sys_ai[0].in_min := 6400;
    sys_ai[0].in_max := 32000;
    sys_ai[0].ai_min := 6300;
    sys_ai[0].ai_max := 32700;
    sys_ai_sp[0].spi.re := sys_ai[0].out_min := 0;
    sys_ai_sp[1].spi.re := sys_ai[0].out_max := 500;
    sys_ai_sp[2].spi.re := sys_ai[0].delta := 2;
    sys_ai_sp[3].spi.re := sys_ai[0].val_fail_min := -26;
    sys_ai_sp[4].spi.re := sys_ai[0].val_fail_max := 90;
    sys_ai_sp[5].spi.re := sys_ai[0].val_warn_min := -26;
    sys_ai_sp[6].spi.re := sys_ai[0].val_warn_max := 80;
    sys_ai_sp[7].spi.re := sys_ai[0].hyst := 0.1;
    sys_ai[0].use_fail_min := True;
    sys_ai[0].use_fail_max := True;
    sys_ai[0].use_warn_min := True;
    sys_ai[0].use_warn_max := True;
    //StrCpyW(ADR(sys_ai[1].name), SIZEOF(sys_ai[1].name), ADR("Напряжение аккумуляторной батареи =24В"));
    //StrCpyW(ADR(sys_ai[1].name), SIZEOF(sys_ai[1].name), ADR("%"));
    sys_ai[1].fail := FALSE;
    sys_ai[1].k := 0.2;
    sys_ai[1].in_min := 6400;
    sys_ai[1].in_max := 32000;
    sys_ai[1].ai_min := 6300;
    sys_ai[1].ai_max := 32700;
    sys_ai_sp[8].spi.re := sys_ai[1].out_min := 0;
    sys_ai_sp[9].spi.re := sys_ai[1].out_max := 50;
    sys_ai_sp[10].spi.re := sys_ai[1].delta := 2;
    sys_ai_sp[11].spi.re := sys_ai[1].val_fail_min := -26;
    sys_ai_sp[12].spi.re := sys_ai[1].val_fail_max := 90;
    sys_ai_sp[13].spi.re := sys_ai[1].val_warn_min := -26;
    sys_ai_sp[14].spi.re := sys_ai[1].val_warn_max := 80;
    sys_ai_sp[15].spi.re := sys_ai[1].hyst := 0.1;
    sys_ai[1].use_fail_min := True;
    sys_ai[1].use_fail_max := True;
    sys_ai[1].use_warn_min := True;
    sys_ai[1].use_warn_max := True;
    //StrCpyW(ADR(sys_ai[2].name), SIZEOF(sys_ai[2].name), ADR("Резерв"));
    //StrCpyW(ADR(sys_ai[2].name), SIZEOF(sys_ai[2].name), ADR("%"));
    sys_ai[2].fail := FALSE;
    sys_ai[2].k := 0.2;
    sys_ai[2].in_min := 6400;
    sys_ai[2].in_max := 32000;
    sys_ai[2].ai_min := 6300;
    sys_ai[2].ai_max := 32700;
    sys_ai_sp[16].spi.re := sys_ai[2].out_min := 0;
    sys_ai_sp[17].spi.re := sys_ai[2].out_max := 100;
    sys_ai_sp[18].spi.re := sys_ai[2].delta := 2;
    sys_ai_sp[19].spi.re := sys_ai[2].val_fail_min := -26;
    sys_ai_sp[20].spi.re := sys_ai[2].val_fail_max := 90;
    sys_ai_sp[21].spi.re := sys_ai[2].val_warn_min := -26;
    sys_ai_sp[22].spi.re := sys_ai[2].val_warn_max := 80;
    sys_ai_sp[23].spi.re := sys_ai[2].hyst := 0.1;
    sys_ai[2].use_fail_min := True;
    sys_ai[2].use_fail_max := True;
    sys_ai[2].use_warn_min := True;
    sys_ai[2].use_warn_max := True;
    //StrCpyW(ADR(sys_ai[3].name), SIZEOF(sys_ai[3].name), ADR("Резерв"));
    //StrCpyW(ADR(sys_ai[3].name), SIZEOF(sys_ai[3].name), ADR("%"));
    sys_ai[3].fail := FALSE;
    sys_ai[3].k := 0.2;
    sys_ai[3].in_min := 6400;
    sys_ai[3].in_max := 32000;
    sys_ai[3].ai_min := 6300;
    sys_ai[3].ai_max := 32700;
    sys_ai_sp[24].spi.re := sys_ai[3].out_min := 0;
    sys_ai_sp[25].spi.re := sys_ai[3].out_max := 100;
    sys_ai_sp[26].spi.re := sys_ai[3].delta := 2;
    sys_ai_sp[27].spi.re := sys_ai[3].val_fail_min := -26;
    sys_ai_sp[28].spi.re := sys_ai[3].val_fail_max := 90;
    sys_ai_sp[29].spi.re := sys_ai[3].val_warn_min := -26;
    sys_ai_sp[30].spi.re := sys_ai[3].val_warn_max := 80;
    sys_ai_sp[31].spi.re := sys_ai[3].hyst := 0.1;
    sys_ai[3].use_fail_min := True;
    sys_ai[3].use_fail_max := True;
    sys_ai[3].use_warn_min := True;
    sys_ai[3].use_warn_max := True;
    //StrCpyW(ADR(sys_ai[4].name), SIZEOF(sys_ai[4].name), ADR("Шунт"));
    //StrCpyW(ADR(sys_ai[4].name), SIZEOF(sys_ai[4].name), ADR("%"));
    sys_ai[4].fail := FALSE;
    sys_ai[4].k := 0.2;
    sys_ai[4].in_min := 6400;
    sys_ai[4].in_max := 32000;
    sys_ai[4].ai_min := 6300;
    sys_ai[4].ai_max := 32700;
    sys_ai_sp[32].spi.re := sys_ai[4].out_min := 0;
    sys_ai_sp[33].spi.re := sys_ai[4].out_max := 100;
    sys_ai_sp[34].spi.re := sys_ai[4].delta := 2;
    sys_ai_sp[35].spi.re := sys_ai[4].val_fail_min := -26;
    sys_ai_sp[36].spi.re := sys_ai[4].val_fail_max := 90;
    sys_ai_sp[37].spi.re := sys_ai[4].val_warn_min := -26;
    sys_ai_sp[38].spi.re := sys_ai[4].val_warn_max := 80;
    sys_ai_sp[39].spi.re := sys_ai[4].hyst := 0.1;
    sys_ai[4].use_fail_min := True;
    sys_ai[4].use_fail_max := True;
    sys_ai[4].use_warn_min := True;
    sys_ai[4].use_warn_max := True;
    //StrCpyW(ADR(sys_ai[5].name), SIZEOF(sys_ai[5].name), ADR("Потенциал трубы"));
    //StrCpyW(ADR(sys_ai[5].name), SIZEOF(sys_ai[5].name), ADR("%"));
    sys_ai[5].fail := FALSE;
    sys_ai[5].k := 0.2;
    sys_ai[5].in_min := 6400;
    sys_ai[5].in_max := 32000;
    sys_ai[5].ai_min := 6300;
    sys_ai[5].ai_max := 32700;
    sys_ai_sp[40].spi.re := sys_ai[5].out_min := 0;
    sys_ai_sp[41].spi.re := sys_ai[5].out_max := 100;
    sys_ai_sp[42].spi.re := sys_ai[5].delta := 2;
    sys_ai_sp[43].spi.re := sys_ai[5].val_fail_min := -26;
    sys_ai_sp[44].spi.re := sys_ai[5].val_fail_max := 90;
    sys_ai_sp[45].spi.re := sys_ai[5].val_warn_min := -26;
    sys_ai_sp[46].spi.re := sys_ai[5].val_warn_max := 80;
    sys_ai_sp[47].spi.re := sys_ai[5].hyst := 0.1;
    sys_ai[5].use_fail_min := True;
    sys_ai[5].use_fail_max := True;
    sys_ai[5].use_warn_min := True;
    sys_ai[5].use_warn_max := True;
    //StrCpyW(ADR(sys_ai[6].name), SIZEOF(sys_ai[6].name), ADR("Напряжение СКЗ"));
    //StrCpyW(ADR(sys_ai[6].name), SIZEOF(sys_ai[6].name), ADR("%"));
    sys_ai[6].fail := FALSE;
    sys_ai[6].k := 0.2;
    sys_ai[6].in_min := 6400;
    sys_ai[6].in_max := 32000;
    sys_ai[6].ai_min := 6300;
    sys_ai[6].ai_max := 32700;
    sys_ai_sp[48].spi.re := sys_ai[6].out_min := 0;
    sys_ai_sp[49].spi.re := sys_ai[6].out_max := 100;
    sys_ai_sp[50].spi.re := sys_ai[6].delta := 2;
    sys_ai_sp[51].spi.re := sys_ai[6].val_fail_min := -26;
    sys_ai_sp[52].spi.re := sys_ai[6].val_fail_max := 90;
    sys_ai_sp[53].spi.re := sys_ai[6].val_warn_min := -26;
    sys_ai_sp[54].spi.re := sys_ai[6].val_warn_max := 80;
    sys_ai_sp[55].spi.re := sys_ai[6].hyst := 0.1;
    sys_ai[6].use_fail_min := True;
    sys_ai[6].use_fail_max := True;
    sys_ai[6].use_warn_min := True;
    sys_ai[6].use_warn_max := True;
    //StrCpyW(ADR(sys_ai[7].name), SIZEOF(sys_ai[7].name), ADR("Термосопротивление"));
    //StrCpyW(ADR(sys_ai[7].name), SIZEOF(sys_ai[7].name), ADR("%"));
    sys_ai[7].fail := FALSE;
    sys_ai[7].k := 0.2;
    sys_ai[7].in_min := 6400;
    sys_ai[7].in_max := 32000;
    sys_ai[7].ai_min := 6300;
    sys_ai[7].ai_max := 32700;
    sys_ai_sp[56].spi.re := sys_ai[7].out_min := 0;
    sys_ai_sp[57].spi.re := sys_ai[7].out_max := 100;
    sys_ai_sp[58].spi.re := sys_ai[7].delta := 2;
    sys_ai_sp[59].spi.re := sys_ai[7].val_fail_min := -26;
    sys_ai_sp[60].spi.re := sys_ai[7].val_fail_max := 90;
    sys_ai_sp[61].spi.re := sys_ai[7].val_warn_min := -26;
    sys_ai_sp[62].spi.re := sys_ai[7].val_warn_max := 80;
    sys_ai_sp[63].spi.re := sys_ai[7].hyst := 0.1;
    sys_ai[7].use_fail_min := True;
    sys_ai[7].use_fail_max := True;
    sys_ai[7].use_warn_min := True;
    sys_ai[7].use_warn_max := True;
    //StrCpyW(ADR(sys_ai[8].name), SIZEOF(sys_ai[8].name), ADR("Температура газа после крана № 388.7"));
    //StrCpyW(ADR(sys_ai[8].name), SIZEOF(sys_ai[8].name), ADR("%"));
    sys_ai[8].fail := FALSE;
    sys_ai[8].k := 0.2;
    sys_ai[8].in_min := 6400;
    sys_ai[8].in_max := 32000;
    sys_ai[8].ai_min := 6300;
    sys_ai[8].ai_max := 32700;
    sys_ai_sp[64].spi.re := sys_ai[8].out_min := 0;
    sys_ai_sp[65].spi.re := sys_ai[8].out_max := 100;
    sys_ai_sp[66].spi.re := sys_ai[8].delta := 2;
    sys_ai_sp[67].spi.re := sys_ai[8].val_fail_min := -26;
    sys_ai_sp[68].spi.re := sys_ai[8].val_fail_max := 90;
    sys_ai_sp[69].spi.re := sys_ai[8].val_warn_min := -26;
    sys_ai_sp[70].spi.re := sys_ai[8].val_warn_max := 80;
    sys_ai_sp[71].spi.re := sys_ai[8].hyst := 0.1;
    sys_ai[8].use_fail_min := True;
    sys_ai[8].use_fail_max := True;
    sys_ai[8].use_warn_min := True;
    sys_ai[8].use_warn_max := True;
    //StrCpyW(ADR(sys_ai[9].name), SIZEOF(sys_ai[9].name), ADR("Температура грунта"));
    //StrCpyW(ADR(sys_ai[9].name), SIZEOF(sys_ai[9].name), ADR("%"));
    sys_ai[9].fail := FALSE;
    sys_ai[9].k := 0.2;
    sys_ai[9].in_min := 6400;
    sys_ai[9].in_max := 32000;
    sys_ai[9].ai_min := 6300;
    sys_ai[9].ai_max := 32700;
    sys_ai_sp[72].spi.re := sys_ai[9].out_min := 0;
    sys_ai_sp[73].spi.re := sys_ai[9].out_max := 100;
    sys_ai_sp[74].spi.re := sys_ai[9].delta := 2;
    sys_ai_sp[75].spi.re := sys_ai[9].val_fail_min := -26;
    sys_ai_sp[76].spi.re := sys_ai[9].val_fail_max := 90;
    sys_ai_sp[77].spi.re := sys_ai[9].val_warn_min := -26;
    sys_ai_sp[78].spi.re := sys_ai[9].val_warn_max := 80;
    sys_ai_sp[79].spi.re := sys_ai[9].hyst := 0.1;
    sys_ai[9].use_fail_min := True;
    sys_ai[9].use_fail_max := True;
    sys_ai[9].use_warn_min := True;
    sys_ai[9].use_warn_max := True;
    //StrCpyW(ADR(sys_ai[10].name), SIZEOF(sys_ai[10].name), ADR("Давление газа до крана № 388.7"));
    //StrCpyW(ADR(sys_ai[10].name), SIZEOF(sys_ai[10].name), ADR("%"));
    sys_ai[10].fail := FALSE;
    sys_ai[10].k := 0.2;
    sys_ai[10].in_min := 6400;
    sys_ai[10].in_max := 32000;
    sys_ai[10].ai_min := 6300;
    sys_ai[10].ai_max := 32700;
    sys_ai_sp[80].spi.re := sys_ai[10].out_min := 0;
    sys_ai_sp[81].spi.re := sys_ai[10].out_max := 100;
    sys_ai_sp[82].spi.re := sys_ai[10].delta := 2;
    sys_ai_sp[83].spi.re := sys_ai[10].val_fail_min := -26;
    sys_ai_sp[84].spi.re := sys_ai[10].val_fail_max := 90;
    sys_ai_sp[85].spi.re := sys_ai[10].val_warn_min := -26;
    sys_ai_sp[86].spi.re := sys_ai[10].val_warn_max := 80;
    sys_ai_sp[87].spi.re := sys_ai[10].hyst := 0.1;
    sys_ai[10].use_fail_min := True;
    sys_ai[10].use_fail_max := True;
    sys_ai[10].use_warn_min := True;
    sys_ai[10].use_warn_max := True;
    //StrCpyW(ADR(sys_ai[11].name), SIZEOF(sys_ai[11].name), ADR("Давление газа после крана № 388.7"));
    //StrCpyW(ADR(sys_ai[11].name), SIZEOF(sys_ai[11].name), ADR("%"));
    sys_ai[11].fail := FALSE;
    sys_ai[11].k := 0.2;
    sys_ai[11].in_min := 6400;
    sys_ai[11].in_max := 32000;
    sys_ai[11].ai_min := 6300;
    sys_ai[11].ai_max := 32700;
    sys_ai_sp[88].spi.re := sys_ai[11].out_min := 0;
    sys_ai_sp[89].spi.re := sys_ai[11].out_max := 100;
    sys_ai_sp[90].spi.re := sys_ai[11].delta := 2;
    sys_ai_sp[91].spi.re := sys_ai[11].val_fail_min := -26;
    sys_ai_sp[92].spi.re := sys_ai[11].val_fail_max := 90;
    sys_ai_sp[93].spi.re := sys_ai[11].val_warn_min := -26;
    sys_ai_sp[94].spi.re := sys_ai[11].val_warn_max := 80;
    sys_ai_sp[95].spi.re := sys_ai[11].hyst := 0.1;
    sys_ai[11].use_fail_min := True;
    sys_ai[11].use_fail_max := True;
    sys_ai[11].use_warn_min := True;
    sys_ai[11].use_warn_max := True;
    //StrCpyW(ADR(sys_ai[12].name), SIZEOF(sys_ai[12].name), ADR("Давление газа в аккумуляторе импульчного газа"));
    //StrCpyW(ADR(sys_ai[12].name), SIZEOF(sys_ai[12].name), ADR("%"));
    sys_ai[12].fail := FALSE;
    sys_ai[12].k := 0.2;
    sys_ai[12].in_min := 6400;
    sys_ai[12].in_max := 32000;
    sys_ai[12].ai_min := 6300;
    sys_ai[12].ai_max := 32700;
    sys_ai_sp[96].spi.re := sys_ai[12].out_min := 0;
    sys_ai_sp[97].spi.re := sys_ai[12].out_max := 100;
    sys_ai_sp[98].spi.re := sys_ai[12].delta := 2;
    sys_ai_sp[99].spi.re := sys_ai[12].val_fail_min := -26;
    sys_ai_sp[100].spi.re := sys_ai[12].val_fail_max := 90;
    sys_ai_sp[101].spi.re := sys_ai[12].val_warn_min := -26;
    sys_ai_sp[102].spi.re := sys_ai[12].val_warn_max := 80;
    sys_ai_sp[103].spi.re := sys_ai[12].hyst := 0.1;
    sys_ai[12].use_fail_min := True;
    sys_ai[12].use_fail_max := True;
    sys_ai[12].use_warn_min := True;
    sys_ai[12].use_warn_max := True;
    //StrCpyW(ADR(sys_ai[13].name), SIZEOF(sys_ai[13].name), ADR("Температура воздуха в блок-боксе КП ТМ"));
    //StrCpyW(ADR(sys_ai[13].name), SIZEOF(sys_ai[13].name), ADR("%"));
    sys_ai[13].fail := FALSE;
    sys_ai[13].k := 0.2;
    sys_ai[13].in_min := 6400;
    sys_ai[13].in_max := 32000;
    sys_ai[13].ai_min := 6300;
    sys_ai[13].ai_max := 32700;
    sys_ai_sp[104].spi.re := sys_ai[13].out_min := 0;
    sys_ai_sp[105].spi.re := sys_ai[13].out_max := 100;
    sys_ai_sp[106].spi.re := sys_ai[13].delta := 2;
    sys_ai_sp[107].spi.re := sys_ai[13].val_fail_min := -26;
    sys_ai_sp[108].spi.re := sys_ai[13].val_fail_max := 90;
    sys_ai_sp[109].spi.re := sys_ai[13].val_warn_min := -26;
    sys_ai_sp[110].spi.re := sys_ai[13].val_warn_max := 80;
    sys_ai_sp[111].spi.re := sys_ai[13].hyst := 0.1;
    sys_ai[13].use_fail_min := True;
    sys_ai[13].use_fail_max := True;
    sys_ai[13].use_warn_min := True;
    sys_ai[13].use_warn_max := True;
    //StrCpyW(ADR(sys_ai[14].name), SIZEOF(sys_ai[14].name), ADR("Температура наружнего воздуха"));
    //StrCpyW(ADR(sys_ai[14].name), SIZEOF(sys_ai[14].name), ADR("%"));
    sys_ai[14].fail := FALSE;
    sys_ai[14].k := 0.2;
    sys_ai[14].in_min := 6400;
    sys_ai[14].in_max := 32000;
    sys_ai[14].ai_min := 6300;
    sys_ai[14].ai_max := 32700;
    sys_ai_sp[112].spi.re := sys_ai[14].out_min := 0;
    sys_ai_sp[113].spi.re := sys_ai[14].out_max := 100;
    sys_ai_sp[114].spi.re := sys_ai[14].delta := 2;
    sys_ai_sp[115].spi.re := sys_ai[14].val_fail_min := -26;
    sys_ai_sp[116].spi.re := sys_ai[14].val_fail_max := 90;
    sys_ai_sp[117].spi.re := sys_ai[14].val_warn_min := -26;
    sys_ai_sp[118].spi.re := sys_ai[14].val_warn_max := 80;
    sys_ai_sp[119].spi.re := sys_ai[14].hyst := 0.1;
    sys_ai[14].use_fail_min := True;
    sys_ai[14].use_fail_max := True;
    sys_ai[14].use_warn_min := True;
    sys_ai[14].use_warn_max := True;
    //StrCpyW(ADR(sys_ai[15].name), SIZEOF(sys_ai[15].name), ADR("Резерв"));
    //StrCpyW(ADR(sys_ai[15].name), SIZEOF(sys_ai[15].name), ADR("%"));
    sys_ai[15].fail := FALSE;
    sys_ai[15].k := 0.2;
    sys_ai[15].in_min := 6400;
    sys_ai[15].in_max := 32000;
    sys_ai[15].ai_min := 6300;
    sys_ai[15].ai_max := 32700;
    sys_ai_sp[120].spi.re := sys_ai[15].out_min := 0;
    sys_ai_sp[121].spi.re := sys_ai[15].out_max := 100;
    sys_ai_sp[122].spi.re := sys_ai[15].delta := 2;
    sys_ai_sp[123].spi.re := sys_ai[15].val_fail_min := -26;
    sys_ai_sp[124].spi.re := sys_ai[15].val_fail_max := 90;
    sys_ai_sp[125].spi.re := sys_ai[15].val_warn_min := -26;
    sys_ai_sp[126].spi.re := sys_ai[15].val_warn_max := 80;
    sys_ai_sp[127].spi.re := sys_ai[15].hyst := 0.1;
    sys_ai[15].use_fail_min := True;
    sys_ai[15].use_fail_max := True;
    sys_ai[15].use_warn_min := True;
    sys_ai[15].use_warn_max := True;
    
    
    StrCpyW(ADR(sys_valve[0].name), SIZEOF(sys_valve[0].name), ADR("Кран № 388.7 (№1)"));
    sys_valve[0].type_valve := 0;
    sys_valve[0].type_sol := 1;
    sys_valve[0].type_cv := 1;
    sys_valve[0].sp.cvw := 3;
    sys_valve_sp[0].spi.ui := sys_valve[0].sp.start := 5;
    sys_valve_sp[1].spi.ui := sys_valve[0].sp.moving := 30;
    sys_valve_sp[2].spi.ui := sys_valve[0].sp.press := 3;
    sys_valve[0].sp.imit := 3;
    sys_valve[0].sp.sol := 1;
    StrCpyW(ADR(sys_valve[1].name), SIZEOF(sys_valve[1].name), ADR("Резервный кран (№2)"));
    sys_valve[1].type_valve := 0;
    sys_valve[1].type_sol := 1;
    sys_valve[1].type_cv := 1;
    sys_valve[1].sp.cvw := 3;
    sys_valve_sp[3].spi.ui := sys_valve[1].sp.start := 5;
    sys_valve_sp[4].spi.ui := sys_valve[1].sp.moving := 30;
    sys_valve_sp[5].spi.ui := sys_valve[1].sp.press := 3;
    sys_valve[1].sp.imit := 3;
    sys_valve[1].sp.sol := 1;
    
// [N_stop, N_valve, N_step]
    
    
    station.cfg.conf_valve_dist := True;
    station.num_di_valve_dist := 13;
    station.cfg.conf_valve_cv := True;
    station.num_do_valve_cv := 7;
    station.cfg.conf_unit_dist := False;
    station.cfg.conf_unit_cv := False;
    station.cfg.conf_sound_block := False;
    station.cfg.conf_ack := False;
    station.cfg.conf_stop_1 := False;
    station.cfg.conf_stop_2 := False;
    station.cfg.conf_sound := False;
    station.cfg.conf_test_sound := False;
    station.cfg.conf_alarm := False;
    station.cfg.conf_test_alarm := False;
    station.cfg.conf_fail := False;
    station.cfg.conf_warn := False;
    station.cfg.conf_fire := False;
    station.cfg.conf_gas := False;
    station.cfg.conf_lamps := False;
    station.cfg.conf_warn_is_alarm := False;
    
    StrCpyA(ADR(DaemonIP.port_cfg_eth[0].host), SIZEOF(DaemonIP.port_cfg_eth[0].host), ADR('172.16.26.30'));
    DaemonIP.port_cfg_eth[0].port := 502;
    DaemonIP.port_cfg_eth[0].enable := True;
    
    DaemonSerial.port_cfg_serial[0].port := 2;
    DaemonSerial.port_cfg_serial[0].portMode := RLTM.SERIAL_PORT_MODE.BINARY;
    DaemonSerial.port_cfg_serial[0].baudrate := 115200;
    DaemonSerial.port_cfg_serial[0].dataBits := RLTM.SERIAL_DATA_BITS.EIGHT_BITS;
    DaemonSerial.port_cfg_serial[0].parity := RLTM.SERIAL_PARITY.PARITY_NONE;
    DaemonSerial.port_cfg_serial[0].stopBits := RLTM.SERIAL_STOP_BITS.ONE_BIT;
    DaemonSerial.port_cfg_serial[0].enable := True;
    DaemonSerial.port_cfg_serial[1].port := 100;
    DaemonSerial.port_cfg_serial[1].portMode := RLTM.SERIAL_PORT_MODE.BINARY;
    DaemonSerial.port_cfg_serial[1].baudrate := 115200;
    DaemonSerial.port_cfg_serial[1].dataBits := RLTM.SERIAL_DATA_BITS.EIGHT_BITS;
    DaemonSerial.port_cfg_serial[1].parity := RLTM.SERIAL_PARITY.PARITY_NONE;
    DaemonSerial.port_cfg_serial[1].stopBits := RLTM.SERIAL_STOP_BITS.ONE_BIT;
    DaemonSerial.port_cfg_serial[1].enable := True;
    DaemonSerial.port_cfg_serial[2].port := 101;
    DaemonSerial.port_cfg_serial[2].portMode := RLTM.SERIAL_PORT_MODE.BINARY;
    DaemonSerial.port_cfg_serial[2].baudrate := 115200;
    DaemonSerial.port_cfg_serial[2].dataBits := RLTM.SERIAL_DATA_BITS.EIGHT_BITS;
    DaemonSerial.port_cfg_serial[2].parity := RLTM.SERIAL_PARITY.PARITY_NONE;
    DaemonSerial.port_cfg_serial[2].stopBits := RLTM.SERIAL_STOP_BITS.ONE_BIT;
    DaemonSerial.port_cfg_serial[2].enable := True;
    DaemonSerial.port_cfg_serial[3].port := 102;
    DaemonSerial.port_cfg_serial[3].portMode := RLTM.SERIAL_PORT_MODE.BINARY;
    DaemonSerial.port_cfg_serial[3].baudrate := 115200;
    DaemonSerial.port_cfg_serial[3].dataBits := RLTM.SERIAL_DATA_BITS.EIGHT_BITS;
    DaemonSerial.port_cfg_serial[3].parity := RLTM.SERIAL_PARITY.PARITY_NONE;
    DaemonSerial.port_cfg_serial[3].stopBits := RLTM.SERIAL_STOP_BITS.ONE_BIT;
    DaemonSerial.port_cfg_serial[3].enable := True;
    DaemonSerial.port_cfg_serial[4].port := 103;
    DaemonSerial.port_cfg_serial[4].portMode := RLTM.SERIAL_PORT_MODE.BINARY;
    DaemonSerial.port_cfg_serial[4].baudrate := 115200;
    DaemonSerial.port_cfg_serial[4].dataBits := RLTM.SERIAL_DATA_BITS.EIGHT_BITS;
    DaemonSerial.port_cfg_serial[4].parity := RLTM.SERIAL_PARITY.PARITY_NONE;
    DaemonSerial.port_cfg_serial[4].stopBits := RLTM.SERIAL_STOP_BITS.ONE_BIT;
    DaemonSerial.port_cfg_serial[4].enable := True;
    DaemonSerial.port_cfg_serial[5].port := 104;
    DaemonSerial.port_cfg_serial[5].portMode := RLTM.SERIAL_PORT_MODE.BINARY;
    DaemonSerial.port_cfg_serial[5].baudrate := 115200;
    DaemonSerial.port_cfg_serial[5].dataBits := RLTM.SERIAL_DATA_BITS.EIGHT_BITS;
    DaemonSerial.port_cfg_serial[5].parity := RLTM.SERIAL_PARITY.PARITY_NONE;
    DaemonSerial.port_cfg_serial[5].stopBits := RLTM.SERIAL_STOP_BITS.ONE_BIT;
    DaemonSerial.port_cfg_serial[5].enable := True;
    DaemonSerial.port_cfg_serial[6].port := 105;
    DaemonSerial.port_cfg_serial[6].portMode := RLTM.SERIAL_PORT_MODE.BINARY;
    DaemonSerial.port_cfg_serial[6].baudrate := 115200;
    DaemonSerial.port_cfg_serial[6].dataBits := RLTM.SERIAL_DATA_BITS.EIGHT_BITS;
    DaemonSerial.port_cfg_serial[6].parity := RLTM.SERIAL_PARITY.PARITY_NONE;
    DaemonSerial.port_cfg_serial[6].stopBits := RLTM.SERIAL_STOP_BITS.ONE_BIT;
    DaemonSerial.port_cfg_serial[6].enable := True;
END_METHOD

METHOD Init_User
VAR_INPUT
END_VAR
VAR
	i, N: UINT;
END_VAR
END_METHOD

METHOD Cyclic_In
VAR_INPUT
END_VAR
    
    sys_di[0].fail := NOT sys_mod[1].ok;
    sys_di[1].fail := NOT sys_mod[1].ok;
    sys_di[2].fail := NOT sys_mod[1].ok;
    sys_di[3].fail := NOT sys_mod[1].ok;
    sys_di[4].fail := NOT sys_mod[1].ok;
    sys_di[5].fail := NOT sys_mod[1].ok;
    sys_di[6].fail := NOT sys_mod[1].ok;
    sys_di[7].fail := NOT sys_mod[1].ok;
    sys_di[8].fail := NOT sys_mod[1].ok;
    sys_di[9].fail := NOT sys_mod[1].ok;
    sys_di[10].fail := NOT sys_mod[1].ok;
    sys_di[11].fail := NOT sys_mod[1].ok;
    sys_di[12].fail := NOT sys_mod[1].ok;
    sys_di[13].fail := NOT sys_mod[1].ok;
    sys_di[14].fail := NOT sys_mod[1].ok;
    sys_di[15].fail := NOT sys_mod[1].ok;
    sys_di[16].fail := NOT sys_mod[1].ok;
    sys_di[17].fail := NOT sys_mod[1].ok;
    sys_di[18].fail := NOT sys_mod[1].ok;
    sys_di[19].fail := NOT sys_mod[1].ok;
    sys_di[20].fail := NOT sys_mod[1].ok;
    sys_di[21].fail := NOT sys_mod[1].ok;
    sys_di[22].fail := NOT sys_mod[1].ok;
    sys_di[23].fail := NOT sys_mod[1].ok;
    sys_di[24].fail := NOT sys_mod[1].ok;
    sys_di[25].fail := NOT sys_mod[1].ok;
    sys_di[26].fail := NOT sys_mod[1].ok;
    sys_di[27].fail := NOT sys_mod[1].ok;
    sys_di[28].fail := NOT sys_mod[1].ok;
    sys_di[29].fail := NOT sys_mod[1].ok;
    sys_di[30].fail := NOT sys_mod[1].ok;
    sys_di[31].fail := NOT sys_mod[1].ok;
    sys_di[32].fail := NOT sys_mod[2].ok;
    sys_di[33].fail := NOT sys_mod[2].ok;
    sys_di[34].fail := NOT sys_mod[2].ok;
    sys_di[35].fail := NOT sys_mod[2].ok;
    sys_di[36].fail := NOT sys_mod[2].ok;
    sys_di[37].fail := NOT sys_mod[2].ok;
    sys_di[38].fail := NOT sys_mod[2].ok;
    sys_di[39].fail := NOT sys_mod[2].ok;
    sys_di[40].fail := NOT sys_mod[2].ok;
    sys_di[41].fail := NOT sys_mod[2].ok;
    sys_di[42].fail := NOT sys_mod[2].ok;
    sys_di[43].fail := NOT sys_mod[2].ok;
    sys_di[44].fail := NOT sys_mod[2].ok;
    sys_di[45].fail := NOT sys_mod[2].ok;
    sys_di[46].fail := NOT sys_mod[2].ok;
    sys_di[47].fail := NOT sys_mod[2].ok;
    
    sys_ai[0].fail := NOT sys_mod[3].ok;
    sys_ai[1].fail := NOT sys_mod[3].ok;
    sys_ai[2].fail := NOT sys_mod[3].ok;
    sys_ai[3].fail := NOT sys_mod[3].ok;
    sys_ai[4].fail := NOT sys_mod[3].ok;
    sys_ai[5].fail := NOT sys_mod[3].ok;
    sys_ai[6].fail := NOT sys_mod[3].ok;
    sys_ai[7].fail := NOT sys_mod[3].ok;
    sys_ai[8].fail := NOT sys_mod[3].ok;
    sys_ai[9].fail := NOT sys_mod[3].ok;
    sys_ai[10].fail := NOT sys_mod[3].ok;
    sys_ai[11].fail := NOT sys_mod[3].ok;
    sys_ai[12].fail := NOT sys_mod[3].ok;
    sys_ai[13].fail := NOT sys_mod[3].ok;
    sys_ai[14].fail := NOT sys_mod[3].ok;
    sys_ai[15].fail := NOT sys_mod[3].ok;
    
    sys_valve[0].in.di_dist := sys_di[13].ts;
    sys_valve[0].in.di_open := sys_di[0].ts;
    sys_valve[0].in.di_close := sys_di[1].ts;
    sys_valve[0].in.di_cv := sys_di[12].ts;
    sys_valve[0].in.sol_open := sys_di[2].ts;
    sys_valve[0].in.sol_close := sys_di[3].ts;
    sys_valve[1].in.di_dist := sys_di[13].ts;
    sys_valve[1].in.di_open := sys_di[4].ts;
    sys_valve[1].in.di_close := sys_di[5].ts;
    sys_valve[1].in.di_cv := sys_di[12].ts;
    sys_valve[1].in.sol_open := sys_di[6].ts;
    sys_valve[1].in.sol_close := sys_di[7].ts;
END_METHOD

METHOD Cyclic_Main
VAR_INPUT
END_VAR
VAR
	c: BOOL;
	bc, bl: BOOL;
	i: UINT;
END_VAR
bc := FALSE;
i := 0; WHILE i < COUNT_DI DO
	sys_di[i]();
	bc := bc OR sys_di[i].sb;
	i := i + 1;
END_WHILE
station.global_imit_di := bc;

bc := FALSE;
i := 0; WHILE i < COUNT_AI DO
	sys_ai_sp[i*8+0]();
	sys_ai_sp[i*8+1]();
	sys_ai_sp[i*8+2]();
	sys_ai_sp[i*8+3]();
	sys_ai_sp[i*8+4]();
	sys_ai_sp[i*8+5]();
	sys_ai_sp[i*8+6]();
	sys_ai_sp[i*8+7]();
	
	sys_ai[i].out_min := sys_ai_sp[i*8+0].sp.re;
	sys_ai[i].out_max := sys_ai_sp[i*8+1].sp.re;
	sys_ai[i].delta := sys_ai_sp[i*8+2].sp.re;
	sys_ai[i].val_fail_min := sys_ai_sp[i*8+3].sp.re;
	sys_ai[i].val_fail_max := sys_ai_sp[i*8+4].sp.re;
	sys_ai[i].val_warn_min := sys_ai_sp[i*8+5].sp.re;
	sys_ai[i].val_warn_max := sys_ai_sp[i*8+6].sp.re;
	sys_ai[i].hyst := sys_ai_sp[i*8+7].sp.re;
	
	sys_ai[i]();
	bc := bc OR sys_ai[i].sb;
	i := i + 1;
END_WHILE
station.global_imit_ai := bc;


bc := FALSE; bl := FALSE;
i := 0; WHILE i < COUNT_VALVE DO
	sys_valve_sp[i*3+0]();
	sys_valve_sp[i*3+1]();
	sys_valve_sp[i*3+2]();
	sys_valve[i].sp.start := sys_valve_sp[i*3+0].sp.ui;
	sys_valve[i].sp.moving := sys_valve_sp[i*3+1].sp.ui;
	sys_valve[i].sp.press := sys_valve_sp[i*3+2].sp.ui;
	
	c := sys_valve[i].flags.mode_block;
	sys_valve[i]();
	IF c <> sys_valve[i].flags.mode_block THEN	// было изменение?
		sys_valve_m[i].sp0.b := sys_valve[i].flags.mode_block;	// пробуем записать его в память
		sys_valve_m[i].cmd := TRUE;
		sys_valve_m[i]();
		IF sys_valve_m[i].sp.b <> sys_valve[i].flags.mode_block OR sys_valve_m[i].err_write THEN
			sys_valve[i]._set_block(c);			// если маска не записалась или ошибка - взвести флаг
			sys_valve[i]._set_f_block(TRUE);
		END_IF
	END_IF
	bc := bc OR sys_valve[i].flags.cv_fail;
	bl := bl OR sys_valve[i].flags.mode_imit;
	i := i + 1;
END_WHILE
station.fail_valve_cv := bc;
station.global_imit_valve := bl;

bc := FALSE; bl := FALSE;
i := 0; WHILE i < COUNT_STOP DO
	c := sys_stop[i].flags.mode_block;
	sys_stop[i]();
	IF c <> sys_stop[i].flags.mode_block THEN
		sys_stop_m[i].sp0.b := sys_stop[i].flags.mode_block;
		sys_stop_m[i].cmd := TRUE;
		sys_stop_m[i]();
		IF sys_stop_m[i].sp.b <> sys_stop[i].flags.mode_block OR sys_stop_m[i].err_write THEN
			sys_stop[i]._set_block(c);
			sys_stop[i]._set_f_block(TRUE);
		END_IF
	END_IF
	bc := bc OR sys_stop[i].flags.executing;
	IF station.mode = en_stt_mode.MODE_AUTO AND (sys_stop[i].status = RLTAB.en_stop_step.AUTO_COMPLETED) AND sys_stop[i].cfg.1 (*stop_auto_after*) THEN
		station.cmd.mode_auto_reset := TRUE;
	END_IF
	i := i + 1;
END_WHILE
station.global_stop := bc;

bc := FALSE; bl := FALSE;
i := 0; WHILE i < COUNT_UNIT DO
	sys_unit_sp[i*2+0]();
	sys_unit_sp[i*2+1]();
	sys_unit[i].sp.switch := sys_unit_sp[i*2+0].sp.ui;
	sys_unit[i].sp.work := sys_unit_sp[i*2+1].sp.ui;
	
